# B&R Automation Studio project VisionSample (part 3)

#### brdkFile_func.h - Header for internal functions for library.
```c
#ifndef BRDK_FILE_FUNCS
#define BRDK_FILE_FUNCS 1

#include <brdkFile.h>
#include <bur/plctypes.h>

#ifdef __cplusplus
	extern "C"
	{
#endif

#ifdef __cplusplus
	};
#endif

#define false 0
#define true 1
#define NULL 0

unsigned long buildParameterString(char* pDrive,char* pPath, char* pDeviceParam);
char* getDrive(brdk_file_drive_typ drive, char* pDrive);
signed long splitFolderPath(char* pDestination, char* pSource);

#endif /* !BRDK_FILE_FUNCS */
```

#### brdkFile_func.c - Internal functions for library.
```c
#include <brdkFile_func.h>

unsigned long buildParameterString(char* pDrive,char* pPath, char* pDeviceParam) {
	brdkStrCpy((unsigned long)pDeviceParam,(unsigned long)"/DEVICE=\"");
	brdkStrCat((unsigned long)pDeviceParam,(unsigned long)pDrive);
	brdkStrCat((unsigned long)pDeviceParam,(unsigned long)"\\");
	if(pPath[0] != 0) {
		brdkStrReplace((unsigned long)pPath,(unsigned long)"/",(unsigned long)"\\");	/* replace any front slah with backslash */
		brdkStrCat((unsigned long)pDeviceParam,(unsigned long)pPath);
	}
	brdkStrCat((unsigned long)pDeviceParam,(unsigned long)"\"");
	return (unsigned long)pDeviceParam;
}

char* getDrive(brdk_file_drive_typ drive, char* pDrive) {
	switch(drive) {
		case C_DRIVE: brdkStrCpy((unsigned long)pDrive,(unsigned long)"C:\\"); break;
		case D_DRIVE: brdkStrCpy((unsigned long)pDrive,(unsigned long)"D:\\"); break;
		case E_DRIVE: brdkStrCpy((unsigned long)pDrive,(unsigned long)"E:\\"); break;
		case F_DRIVE: brdkStrCpy((unsigned long)pDrive,(unsigned long)"F:\\"); break;
		case G_DRIVE: brdkStrCpy((unsigned long)pDrive,(unsigned long)"G:\\"); break;
	}
	return pDrive;
}

signed long splitFolderPath(char* pDestination, char* pSource) {
	int idx = 0;
	signed long pos = -1;
	if(pSource[idx] != 0) {
		pos = brdkStrIndexOf((unsigned long)&pSource[idx],(unsigned long)"\\",BRDK_STR_LEFT_SEARCH);
		if(pos > -1) {
			brdkStrMemCpy((unsigned long)pDestination,(unsigned long)&pSource[idx],(unsigned long)++pos);
			pDestination[pos] = 0;
		}
	}
	return pos;
}
```

- CHANGELOG - brdkFile change log file (not shown)

### revision.txt
```
Version 5.26
- Update to mappVision 4.26
- Changed image request to official function block
- Removed recipe management
- Removed color detection
- Removed optic details
- Removed VC4 support
- Removed TCP proxy task
- Removed function to load VA applications
- Removed function to download images

Version 5.24
- Update to AS 4.12
- Update to mapp 4.24
- Fixed image download node number is not correct
- Removed old routing files
- Changed image update interval to 500ms

Version 5.15
- Update recipe managment to V1.0
- Updated constant for code reader parameter "ParameterMode"
- Fix ViColor
- Make it possible to change connections
- Updated to official 5.15 versions and official lightbar upgrade
- Vi_Optics added

Version 2.3
 - Added RouteInfo_Tool.ps1
 - Added color detection first version
 - Split up main task into main and visu, integrated light task into main and visu
 - Added funkctionality to rotate the image on the main page
 - Click on the image on the main page toggles now the textposition (crosshair-details) from left to right
 - CodeReader and OCR Text will be shown on the main page and saved in SVG file
 - Added proxy task to eliminate routing batch file
 - Added Pixel Counter hardware and code

Version 2.2
- Added new functionality to show images in every size on the webviewer widget on the mainpage
- Improved repetitive mode
- SVG files save now all information. It is possible to click on the crosshairs to show the details
- Added diagnostic data creation
- Updated recipe management
- Changed public arrays start index to 0 to avoid issues with C task
- Added a VC4 visualization
- Added functionality to show the image on the VC4 visualization (documentation still missing)
- After boot the first found light will be selected
- Some additional improvements, code optimizations & bug fixes

Version 2.1
- Simplified and reduced data structures
- Added function to switch vision applications
- Reduced result content to one page
- Simplified and sorted the task Vi_image
- Moved crosshair handling to task Vi_image
- Some bugfixes in task Vi_image
- Updated to official versions

Version 2.0
- Convert data structure to new camera firmware
- Support for multiple camera's
- Recipe managment for loading and saving parameters
- Download camera images directly through web browser
- Cleaned up UI
- Support for external lights
- Sample task for nettime with motion
```

### VisionVariables.var
```iecst
(*-----------------------------------------------------------------------------------------------------------------------------------------*)
(*Global variables for sensor hardware and vision functions*)
VAR
	gBlob : typBlobMain; (*Data that is specific for the blob function*)
	gCodeReader : typCodeReaderMain; (*Data that is specific for the code reader*)
	gMatch : typMatchMain; (*Data that is specific for the match function*)
	gMT : typMTMain; (*Data that is specific for the measurement function*)
	gOCR : typOCRMain; (*Data that is specific for the OCR function*)
	gPixel : typPixelMain; (*Data that is specific for the Pixel Counter function*)
	gVisionImage : typVisionImage; (*Data for image handling*)
	gVisionLight : ARRAY[0..MAX_NUM_LIGHTS] OF typLightMain; (*General Light  functions that are independent from the inspection function*)
	gVisionNettime : typVisionNettime; (*Data for nettime calculation*)
	gVisionSensor : ARRAY[0..MAX_NUM_CAMS] OF typVisionMain; (*General vision functions that are independent from the inspection function*)
	gSelectedSensor : UINT := 1; (*Selected camera node number*)
	gSelectedLight : UINT := 1; (*Selected Light node number*)
	NettimeCurrent_us : DINT; (*Current Powerlink nettime*)
END_VAR
(*-----------------------------------------------------------------------------------------------------------------------------------------*)
(*Global constants*)
VAR CONSTANT
	MAX_NUM_CAMS : UINT := 6; (*Maximum number of camera's*)
	MAX_NUM_LIGHTS : UINT := 5; (*Maximum number of light's*)
	MAX_NUM_RESULTS : UINT := 10; (*Maximum number of results*)
	MAX_NUM_PRODUCTS : UINT := 8; (*Maximum number of products for color detection*)
	MAX_IDX_VA_LIST : UINT := 19; (*Maximum number of entrys in the Vision Application list*)
	CONVERT_CYCLES : UINT := 2000;
	DEVICE_NAME : STRING[40] := 'VisionFileDevice'; (*File device where the images and recipes are stored*)
	NETTIME_DEFAULT_DELAY : UDINT := 30000; (*This delay is used when software trigger is used and nettime is enabled*)
	NETTIME_ENABLE : BOOL := FALSE; (*Enable nettime code, this generates the nettime when using manual triggers*)
	MAX_NUM_CODETYPES : USINT := 69; (*Maximum number of code types*)
END_VAR
VAR
	CodeTypes : {REDUND_UNREPLICABLE} ARRAY[0..MAX_NUM_CODETYPES] OF STRING[80] := ['Auto Identify (0)','2/5 Industrial (1)','2/5 Interleaved (2)','Codebar (3)','Code 32 (4)','Code 39 (5)','Code 93 (6)','Code 128 (7)','MSI (8)','PharmaCode (9)','EAN-8 (10)','EAN-8 Add-On 2 (11)','EAN-8 Add-On 5 (12)','EAN-13 (13)','EAN-13 Add-On 2 (14)','EAN-13 Add-On 5 (15)',4(''),'UPC-A (20)','UPC-A Add-On 2 (21)','UPC-A Add-On 5 (22)','UPC-E (23)','UPC-E Add-On 2 (24)','UPC-E Add-On 5 (25)',4(''),'GS1-128 (30)','GS1 DataBar Omnidirectional (31)','GS1 DataBar Truncated (32)','GS1 DataBar Stacked (33)','GS1 DataBar Stacked Omnidirectional (34)','GS1 DataBar Limited (35)','GS1 DataBar Expanded (36)','GS1 DataBar ExpandedStacked (37)',12(''),'Data Matrix ECC200 (50)','QR Code Model 1 (51)','QR Code Model 2 (52)','Micro QRCode (53)','PDF417 (54)','Aztec Code (55)',4(''),'GS1 Data Matrix (60)','GS1 QR Code Model 1 (61)','GS1 QR Code Model 2 (62)','GS1 Aztec Code (63)',6('')]; (*Codes types for code reading*)
END_VAR
```

### VisionTypes.typ
```iecst
(*-----------------------------------------------------------------------------------------------------------------------------------------*)
(*General vision structures*)

TYPE
	typVisionMain : 	STRUCT
		CMD : typVisionCommand;
		CFG : typVisionConfig;
		DAT : typVisionData;
		HW : typVisionHW;
	END_STRUCT;
	typVisionCommand : 	STRUCT
		ImageTrigger : BOOL;
		ImageTriggerReset : BOOL;
		AutoSetupStartStop : BOOL;
	END_STRUCT;
	typVisionConfig : 	STRUCT
		VisionFunction : enumVisionFunction;
		PowerlinkNode : USINT;
		DataStructure : UDINT;
		ComponentLink : ViComponentType;
		ResolutionWidth_X : UINT; (*Nr of sensor pixels in x direction (width). Is always bigger than height*)
		ResolutionHeight_Y : UINT; (*Nr of sensor pixels in y direction (height). Is always smaller than width*)
	END_STRUCT;
	typVisionData : 	STRUCT
		Enable : BOOL := FALSE;
		MaxItemCnt : USINT := 10;
		NettimeDelay : DINT;
		Timeout : UINT := 5000;
		Gain : USINT;
		Focus : UINT;
		Exposure : UDINT;
		FlashColor : USINT := 1;
		FlashSegment : USINT := 15;
		LedColor : USINT;
		IRFilter : BOOL;
		OffsetROIX : DINT;
		OffsetROIY : DINT;
		OffsetROIRotationCenterX : DINT;
		OffsetROIRotationCenterY : DINT;
		OffsetROIOrientation : INT;
		ChromaticLock : BOOL;
		Alignment : USINT;
		AutoSetupGain : USINT;
		AutoSetupFocus : UINT;
		AutoSetupExposure : UDINT;
		AcquisitionAcceptedCnt : USINT;
		AcquisitionCompletedCnt : USINT;
		AcquisitionFailedCnt : USINT;
		LightWarningCnt : USINT;
		ImageProcessingError : UINT;
		ImageProcessingActive : BOOL;
		ImageNettime : DINT;
		ProcessingTimeCamera : UINT;
		ProcessingTimeFunction : UINT;
		ResultCnt : USINT;
		CockpitIsActive : BOOL;
		Status : UDINT;
		StatusText : STRING[30];
		Active : BOOL;
	END_STRUCT;
	typVisionHW : 	STRUCT
		Connected : BOOL;
		Ready : BOOL;
		DigitalInput01 : BOOL;
		DigitalOutput01 : BOOL;
		DigitalOutputStatus01 : BOOL;
		DigitalOutput02 : BOOL;
		DigitalOutputStatus02 : BOOL;
		SerialNumber : UDINT;
		ID : UDINT;
		Variant : UDINT;
		Firmware : UDINT;
		Undervoltage : BOOL;
		Temperature : SINT;
	END_STRUCT;
	enumVisionFunction :
		(
		enumFunctionNone,
		enumBlob,
		enumCoderReader,
		enumMatch,
		enumMeasurement,
		enumOCR,
		enumPixelCounter
		);
END_TYPE

(*-----------------------------------------------------------------------------------------------------------------------------------------*)
(*General Light structures*)

TYPE
	typLightMain : 	STRUCT
		CMD : typLightCommand;
		CFG : typLightConfig;
		DAT : typLightData;
		HW : typLightHW;
	END_STRUCT;
	typLightCommand : 	STRUCT
		FlashTrigger : BOOL;
		FlashTriggerReset : BOOL;
	END_STRUCT;
	typLightConfig : 	STRUCT
		LightType : enumLightType;
		PowerlinkNode : USINT;
	END_STRUCT;
	typLightData : 	STRUCT
		Enable : USINT := 1;
		FlashColor : USINT := 1;
		FlashSegment : UINT := 15;
		Exposure : UDINT := 200;
		SetAngle : UINT;
		Timeout : UINT := 5000;
		NettimeDelay : DINT;
		FlashAcceptedCnt : USINT;
		FlashCompletedCnt : USINT;
		FlashFailedCnt : USINT;
		Status : UDINT;
	END_STRUCT;
	typLightHW : 	STRUCT
		Connected : BOOL;
		Ready : BOOL;
		SerialNumber : UDINT;
		ID : UDINT;
		Variant : UDINT;
		Firmware : UDINT;
		TemperatureLED : SINT;
		TemperatureControllerBoard : SINT;
		WarningCnt : USINT;
	END_STRUCT;
	enumLightType :
		(
		enumLightNone,
		enumBacklight,
		enumLightbar
		);
END_TYPE

(*-----------------------------------------------------------------------------------------------------------------------------------------*)
(*General nettime structures*)

TYPE
	typVisionNettime : 	STRUCT
		CMD : typNettimeCommand;
		CFG : typNettimeConfig;
		DAT : typNettimeData;
	END_STRUCT;
	typNettimeCommand : 	STRUCT
		Activate : BOOL;
	END_STRUCT;
	typNettimeConfig : 	STRUCT
		AxisPeriod : LREAL; (*Units when period repeats*)
		AxisPositionTrigger : LREAL; (*Position in the period where trigger is fired*)
		AxisPositionDelay_Cycles : LREAL; (*Delay in PLK cycles for the read position from drive*)
		VisionPreTrigger_Cycles : DINT; (*Number of powerlink cycles the trigger has to be send ahead*)
	END_STRUCT;
	typNettimeData : 	STRUCT
		NettimeNext_us : DINT; (*Calculated nettime for next trigger*)
		NettimeDelta_us : DINT; (*Difference between current nettime and calculated nettime for the camera trigger*)
		AxisPosition : LREAL; (*Current axis position*)
		AxisVelocity : LREAL; (*Current axis position*)
		AxisInVelocity : BOOL; (*Indicates that the axis is moving at speed*)
		Overflow : DINT; (*Counts up when a trigger could not be set on time*)
	END_STRUCT;
END_TYPE

(*-----------------------------------------------------------------------------------------------------------------------------------------*)
(*Image upload structures*)

TYPE
	typVisionImage : 	STRUCT
		CMD : typVisionImageCommand;
		CFG : typVisionImageConfig;
		DAT : typVisionImageData;
	END_STRUCT;
	typVisionImageCommand : 	STRUCT
		CreateDir : BOOL;
		DeleteDir : BOOL;
		DeleteImage : BOOL;
		GetImage : BOOL;
		SaveImage : BOOL;
		Refresh : BOOL;
		ResetError : BOOL;
	END_STRUCT;
	typVisionImageConfig : 	STRUCT
		FileDevice : STRING[80];
		FileName : STRING[80];
		DirName : STRING[80];
		ComponentLink : ViComponentType;
	END_STRUCT;
	typVisionImageData : 	STRUCT
		ImagesList : ARRAY[0..19]OF STRING[80];
		ImageSelected : STRING[80];
		ImagePath : STRING[80];
		ImageLast : STRING[80];
		Crosshair : ARRAY[1..MAX_NUM_RESULTS]OF typVisionImageDataCrosshair;
		Status : DINT;
	END_STRUCT;
	typVisionImageDataCrosshair : 	STRUCT
		CrosshairX : REAL;
		CrosshairY : REAL;
		CrosshairRotate : REAL;
		Text : STRING[1000];
	END_STRUCT;
END_TYPE

(*-----------------------------------------------------------------------------------------------------------------------------------------*)
(*Vision specific structures*)

TYPE
	typCodeReaderMain : 	STRUCT  (*Code reader structures*)
		CodeType : USINT;
		GradingEnable : BOOL;
		RobustnessEnable : BOOL;
		ParameterMode : USINT;
		ParameterOptimization : USINT;
		BarcodeText : ARRAY[1..MAX_NUM_RESULTS]OF STRING[100];
		BarcodeType : ARRAY[1..MAX_NUM_RESULTS]OF USINT;
		PositionX : ARRAY[1..MAX_NUM_RESULTS]OF DINT;
		PositionY : ARRAY[1..MAX_NUM_RESULTS]OF DINT;
		Orientation : ARRAY[1..MAX_NUM_RESULTS]OF INT;
		Grading : ARRAY[1..MAX_NUM_RESULTS]OF SINT;
		EnhancedGrading : ARRAY[1..23]OF USINT;
	END_STRUCT;
	typBlobMain : 	STRUCT  (*Blob function structures*)
		RegionalFeature : BOOL;
		EnhancedBlobInformation : BOOL := FALSE;
		ModelNumber : ARRAY[1..MAX_NUM_RESULTS]OF USINT;
		Clipped : ARRAY[1..MAX_NUM_RESULTS]OF BOOL;
		Area : ARRAY[1..MAX_NUM_RESULTS]OF UDINT;
		PositionX : ARRAY[1..MAX_NUM_RESULTS]OF DINT;
		PositionY : ARRAY[1..MAX_NUM_RESULTS]OF DINT;
		Orientation : ARRAY[1..MAX_NUM_RESULTS]OF INT;
		MeanGrayValue : ARRAY[1..MAX_NUM_RESULTS]OF USINT;
		Length : ARRAY[1..MAX_NUM_RESULTS]OF UDINT;
		Width : ARRAY[1..MAX_NUM_RESULTS]OF UDINT;
	END_STRUCT;
	typMatchMain : 	STRUCT  (*Match function structures*)
		MinScore : USINT := 70;
		MaxOverlap : USINT;
		ModelNumber : ARRAY[1..MAX_NUM_RESULTS]OF USINT;
		Score : ARRAY[1..MAX_NUM_RESULTS]OF USINT;
		PositionX : ARRAY[1..MAX_NUM_RESULTS]OF DINT;
		PositionY : ARRAY[1..MAX_NUM_RESULTS]OF DINT;
		Orientation : ARRAY[1..MAX_NUM_RESULTS]OF INT;
		Scale : ARRAY[1..MAX_NUM_RESULTS]OF USINT;
		RotCenterX : ARRAY[1..MAX_NUM_RESULTS]OF DINT;
		RotCenterY : ARRAY[1..MAX_NUM_RESULTS]OF DINT;
	END_STRUCT;
	typOCRMain : 	STRUCT  (*OCR function structures*)
		ParameterMode : USINT;
		GradingEnable : BOOL;
		Text : ARRAY[1..MAX_NUM_RESULTS]OF STRING[50];
		Grading : ARRAY[1..MAX_NUM_RESULTS]OF USINT;
		PositionX : ARRAY[1..MAX_NUM_RESULTS]OF DINT;
		PositionY : ARRAY[1..MAX_NUM_RESULTS]OF DINT;
		Orientation : ARRAY[1..MAX_NUM_RESULTS]OF INT;
	END_STRUCT;
	typPixelMain : 	STRUCT  (*OCR function structures*)
		EnhancedPixelCounterInformation : BOOL := FALSE;
		ModelNumber : ARRAY[1..MAX_NUM_RESULTS]OF USINT;
		NumPixels : ARRAY[1..MAX_NUM_RESULTS]OF UDINT;
		MinGray : ARRAY[1..MAX_NUM_RESULTS]OF USINT;
		MaxGray : ARRAY[1..MAX_NUM_RESULTS]OF USINT;
		MeanGray : ARRAY[1..MAX_NUM_RESULTS]OF UINT;
		DeviationGray : ARRAY[1..MAX_NUM_RESULTS]OF UINT;
		MedianGray : ARRAY[1..MAX_NUM_RESULTS]OF USINT;
		ModelArea : ARRAY[1..MAX_NUM_RESULTS]OF UDINT;
		NumConnectedComponents : ARRAY[1..MAX_NUM_RESULTS]OF UINT;
		PositionX : ARRAY[1..MAX_NUM_RESULTS]OF DINT;
		PositionY : ARRAY[1..MAX_NUM_RESULTS]OF DINT;
	END_STRUCT;
	typMTMain : 	STRUCT  (*MT function structures*)
		UseResultAsXY : BOOL;
		ParameterMode : USINT;
		Result : ARRAY[1..MAX_NUM_RESULTS]OF DINT;
	END_STRUCT;
END_TYPE
```

### Program Logical/Vision/Vi_main (IEC)

#### Main.st - Init, cyclic, exit code
```iecst
// --------------------------------------------------------------------------------------------------------------------
// General vision task. This is a support task for the mappVision. The following functions are implemneted
// - Translate some values in text messages
// - Reset camera trigger when inspection is finsihed
// - Load vision application
// - Save diagnostic data
// Version 2.x (Check revision history for details)
// --------------------------------------------------------------------------------------------------------------------
PROGRAM _INIT

END_PROGRAM

// -----------------------------------------------------------------------------------------------------------
// Cyclic part
// -----------------------------------------------------------------------------------------------------------
PROGRAM _CYCLIC
	// -----------------------------------------------------------------------------------------------------------
	// Translate camera status in readable text
	// -----------------------------------------------------------------------------------------------------------
	IF gVisionSensor[idSensor].DAT.Status = 0 THEN
		gVisionSensor[idSensor].DAT.StatusText := 'Ready';
	ELSIF gVisionSensor[idSensor].DAT.Status = 16#00000001 THEN
		gVisionSensor[idSensor].DAT.StatusText := 'Image acquisition';
	ELSIF gVisionSensor[idSensor].DAT.Status = 16#00000002 THEN
		gVisionSensor[idSensor].DAT.StatusText := 'Waiting trigger';
	ELSIF gVisionSensor[idSensor].DAT.Status = 16#00000010 THEN
		gVisionSensor[idSensor].DAT.StatusText := 'Searching settings';
	ELSIF gVisionSensor[idSensor].DAT.Status = 16#00000080 THEN
		gVisionSensor[idSensor].DAT.StatusText := 'Setting focus';
	ELSIF gVisionSensor[idSensor].DAT.Status = 16#00000090 THEN
		gVisionSensor[idSensor].DAT.StatusText := 'Searching settings';
	ELSIF gVisionSensor[idSensor].DAT.Status = 16#00000800 THEN
		gVisionSensor[idSensor].DAT.StatusText := 'Cam CPU not ready';
	ELSIF gVisionSensor[idSensor].DAT.Status = 16#00001000 THEN
		gVisionSensor[idSensor].DAT.StatusText := 'Cam sensor not ready';
	ELSIF gVisionSensor[idSensor].DAT.Status = 16#01000000 OR gVisionSensor[idSensor].DAT.Status = 16#02000000 OR gVisionSensor[idSensor].DAT.Status = 16#03000000 THEN
		gVisionSensor[idSensor].DAT.StatusText := 'OS check/update';
	ELSIF gVisionSensor[idSensor].DAT.Status = 16#80000000 THEN
		gVisionSensor[idSensor].DAT.StatusText := 'Vision cockpit active';
	ELSE
		// Display the status in hex format 0x02000800
		gVisionSensor[idSensor].DAT.StatusText := '';
		FOR i := 0 TO 28 BY 4 DO
			gVisionSensor[idSensor].DAT.StatusText := CONCAT(MID(HexTab, 1, LIMIT(1, UDINT_TO_INT((SHR(gVisionSensor[idSensor].DAT.Status, i) AND 16#0000000F) + 1), 16)), gVisionSensor[idSensor].DAT.StatusText);
		END_FOR
		gVisionSensor[idSensor].DAT.StatusText := CONCAT('0x', gVisionSensor[idSensor].DAT.StatusText);
	END_IF

	// -----------------------------------------------------------------------------------------------------------
	// Check if vision cockpit is open
	// -----------------------------------------------------------------------------------------------------------
	gVisionSensor[idSensor].DAT.CockpitIsActive := (gVisionSensor[idSensor].DAT.Status AND 16#8000_0000) > 0;

	// -----------------------------------------------------------------------------------------------------------
	// Auto setup handling
	// -----------------------------------------------------------------------------------------------------------
	IF(gVisionSensor[idSensor].CMD.AutoSetupStartStop AND gVisionSensor[idSensor].DAT.Status <> 0) THEN
		AutoSetupRunning[idSensor] := TRUE;
	ELSIF NOT gVisionSensor[idSensor].CMD.AutoSetupStartStop THEN
		AutoSetupRunning[idSensor] := FALSE;
	END_IF
	IF(gVisionSensor[idSensor].CMD.AutoSetupStartStop AND gVisionSensor[idSensor].DAT.Status = 0 AND AutoSetupRunning[idSensor]) THEN // Setup successfully finished
		gVisionSensor[idSensor].DAT.Gain					:= gVisionSensor[idSensor].DAT.AutoSetupGain;
		gVisionSensor[idSensor].DAT.Focus				:= gVisionSensor[idSensor].DAT.AutoSetupFocus;
		gVisionSensor[idSensor].DAT.Exposure				:= gVisionSensor[idSensor].DAT.AutoSetupExposure;
		gVisionSensor[idSensor].CMD.AutoSetupStartStop	:= FALSE;
		AutoSetupRunning[idSensor]						:= FALSE;
		TON_DelayAfterAutoSetup[idSensor].IN					:= TRUE;
	END_IF
	TON_DelayAfterAutoSetup[idSensor](PT := T#50ms);
	IF TON_DelayAfterAutoSetup[idSensor].Q THEN // After the camera tells it is ready, we need to wait still at least ca 20ms, otherwise it does not accept the trigger
		TON_DelayAfterAutoSetup[idSensor].IN := FALSE;
		IF gVisionSensor[idSensor].HW.Ready AND NOT gVisionSensor[idSensor].DAT.ImageProcessingActive THEN
			IF NETTIME_ENABLE THEN
				gVisionSensor[idSensor].DAT.NettimeDelay := NettimeCurrent_us + NETTIME_DEFAULT_DELAY;
			END_IF
			gVisionSensor[idSensor].CMD.ImageTrigger	:= TRUE;
			gVisionSensor[idSensor].DAT.Active			:= TRUE;
		END_IF
	END_IF

	// -----------------------------------------------------------------------------------------------------------
	// Reset image trigger, reload web page and store image when process is finished
	// -----------------------------------------------------------------------------------------------------------
	IF ((gVisionSensor[idSensor].DAT.AcquisitionCompletedCnt <> AcquisitionCompletedCntOld[idSensor] OR gVisionSensor[idSensor].DAT.AcquisitionFailedCnt <> AcquisitionFailedCntOld[idSensor]) AND NOT gVisionSensor[idSensor].DAT.ImageProcessingActive AND gVisionSensor[idSensor].HW.Ready) THEN
		AcquisitionCompletedCntOld[idSensor]		:= gVisionSensor[idSensor].DAT.AcquisitionCompletedCnt;
		AcquisitionFailedCntOld[idSensor]			:= gVisionSensor[idSensor].DAT.AcquisitionFailedCnt;
		gVisionSensor[idSensor].CMD.ImageTrigger	:= FALSE;
		gVisionSensor[idSensor].DAT.Active			:= FALSE;
	END_IF

	// -----------------------------------------------------------------------------------------------------------
	// Reset trigger when timed out
	// -----------------------------------------------------------------------------------------------------------
	IF gVisionSensor[idSensor].CMD.ImageTrigger THEN
		TriggerTimeoutSensor[idSensor].IN := TRUE;
		TriggerTimeoutSensor[idSensor].PT := REAL_TO_TIME(gVisionSensor[idSensor].DAT.Timeout * 1.25);
		IF TriggerTimeoutSensor[idSensor].Q THEN
			gVisionSensor[idSensor].CMD.ImageTrigger		:= FALSE;
			gVisionSensor[idSensor].CMD.ImageTriggerReset	:= TRUE;
			gVisionSensor[idSensor].DAT.Active				:= FALSE;
		END_IF
	ELSE
		TriggerTimeoutSensor[idSensor].IN := FALSE;
		gVisionSensor[idSensor].CMD.ImageTriggerReset := FALSE;
	END_IF
	TriggerTimeoutSensor[idSensor]();

	// Proceed with next sensor
	idSensor := idSensor + 1;
	IF (idSensor > MAX_NUM_CAMS) THEN
		idSensor := 1;
	END_IF

	// -----------------------------------------------------------------------------------------------------------
	// Reset Light trigger
	// -----------------------------------------------------------------------------------------------------------
	IF (gVisionLight[idLight].DAT.FlashCompletedCnt <> FlashCompletedCntOld[idLight] OR gVisionLight[idLight].DAT.FlashFailedCnt <> FlashFailedCntOld[idLight]) THEN
		FlashCompletedCntOld[idLight]			:= gVisionLight[idLight].DAT.FlashCompletedCnt;
		FlashFailedCntOld[idLight]				:= gVisionLight[idLight].DAT.FlashFailedCnt;
		gVisionLight[idLight].CMD.FlashTrigger	:= FALSE;
	END_IF

	// -----------------------------------------------------------------------------------------------------------
	// Reset trigger when timed out
	// -----------------------------------------------------------------------------------------------------------
	IF gVisionLight[idLight].CMD.FlashTrigger THEN
		TriggerTimeoutLight[idLight].IN := TRUE;
		TriggerTimeoutLight[idLight].PT := REAL_TO_TIME(gVisionLight[idLight].DAT.Timeout * 1.25);
		IF TriggerTimeoutLight[idLight].Q THEN
			gVisionLight[idLight].CMD.FlashTrigger		:= FALSE;
			gVisionLight[idLight].CMD.FlashTriggerReset	:= TRUE;
		END_IF
	ELSE
		TriggerTimeoutLight[idLight].IN := FALSE;
		gVisionLight[idLight].CMD.FlashTriggerReset := FALSE;
	END_IF
	TriggerTimeoutLight[idLight]();

	// Proceed with next light
	idLight := idLight + 1;
	IF (idLight > MAX_NUM_LIGHTS) THEN
		idLight := 1;
	END_IF

END_PROGRAM
```

#### Variables.var - Local variables
```iecst
VAR
	i : UINT;
END_VAR
(*-----------------------------------------------------------------------------------------------------------------------------------------*)
(*Local variables*)
VAR
	idSensor : UINT := 1;
	idLight : UINT := 1;
	TriggerTimeoutSensor : ARRAY[1..MAX_NUM_CAMS] OF TON; (*Disable web reload when timed out*)
	TriggerTimeoutLight : ARRAY[1..MAX_NUM_LIGHTS] OF TON; (*Disable web reload when timed out*)
	AcquisitionFailedCntOld : ARRAY[1..MAX_NUM_CAMS] OF UDINT; (*Old aquisition failed counter*)
	AcquisitionCompletedCntOld : ARRAY[1..MAX_NUM_CAMS] OF UDINT; (*Old aquisition completed counter*)
	AutoSetupRunning : ARRAY[1..MAX_NUM_CAMS] OF BOOL; (*Flag for auto setup running*)
	FlashFailedCntOld : ARRAY[1..MAX_NUM_LIGHTS] OF USINT;
	FlashCompletedCntOld : ARRAY[1..MAX_NUM_LIGHTS] OF USINT;
END_VAR
VAR CONSTANT
	HexTab : STRING[16] := '0123456789ABCDEF';
END_VAR
VAR
	TON_DelayAfterAutoSetup : ARRAY[1..MAX_NUM_CAMS] OF TON;
END_VAR
```

#### Types.typ
```iecst
TYPE
	local_axisTrig_typ : 	STRUCT
		nettimeLastCycle_us : DINT;
		powerlinkCycle_us : DINT;
		axisPositionNow : REAL;
		triggerPosDelta : REAL;
		triggerTimeDelta : DINT; (*In us*)
	END_STRUCT;
	local_typ : 	STRUCT
		path : STRING[100];
		brdkViBase_imgTrigger_0 : brdkViBase_imgTrigger;
		brdkViBase_getCameraInfo_0 : brdkViBase_getCameraInfo;
		mappView : {REDUND_UNREPLICABLE} brdkViImg_mappView;
		viBaseSaveDiagData_0 : ViBaseSaveDiagData;
		fileDelete : FileDelete;
		visionDiagFileDevice : STRING[10];
		viBaseLoadApplication_0 : ViBaseLoadApplication;
		axisTrig : local_axisTrig_typ;
		brdkFileWrite : brdkFileWrite;
		dtNow : DTStructure;
		DTGetTime_0 : DTGetTime;
		tmp2D : brdkViBase_2d_typ;
		strElemId : STRING[80];
		oldIntElemID : USINT;
		elemId : STRING[80];
	END_STRUCT;
	hmi_typ : 	STRUCT
		in : hmi_in_typ;
		out : hmi_out_typ;
	END_STRUCT;
	hmi_out_vf_typ : 	STRUCT
		processingTime : UDINT;
		numResults : USINT;
		crData : ARRAY[0..9]OF STRING[240];
		match : typMatchMain;
		measurement : typMTMain;
		codeReader : typCodeReaderMain;
		ocr : typOCRMain;
		pixelCnt : typPixelMain;
		blob : typBlobMain;
		ocrData : ARRAY[0..9]OF STRING[240];
	END_STRUCT;
	hmi_out_lights_typ : 	STRUCT
		status : brdkViBase_light_hw_status_typ;
		common : brdkViBase_hw_in_common_typ;
		simulated : BOOL;
		connectedText : STRING[20];
		connected : BOOL;
		mappVisionActive : BOOL;
		processing : BOOL;
		ready : BOOL;
		statusText : STRING[50];
		lightType : STRING[20];
		plNodeNr : USINT;
	END_STRUCT;
	hmi_out_camera_typ : 	STRUCT
		simulated : BOOL;
		connectedText : STRING[20];
		connected : BOOL;
		mappVisionActive : BOOL;
		processing : BOOL;
		ready : BOOL;
		statusText : STRING[50];
		plNodeNr : USINT;
		visionFunction : STRING[20];
		processingTime : UDINT;
		opticInfo : brdkViBase_opticInfo_typ;
		common : brdkViBase_hw_in_common_typ;
		hw : brdkViBase_cam_hw_in_status_typ;
	END_STRUCT;
	hmi_out_typ : 	STRUCT
		svgOverlay : STRING[10000];
		wsPort : UINT;
		lights : ARRAY[START_IDX..NUM_LIGHTS]OF hmi_out_lights_typ;
		camera : hmi_out_camera_typ;
		VF : hmi_out_vf_typ;
		status : DINT;
	END_STRUCT;
	hmi_in_cmd_flashSegment_typ : 	STRUCT
		top : BOOL := TRUE;
		bottom : BOOL := TRUE;
		right : BOOL := TRUE;
		left : BOOL := TRUE;
	END_STRUCT;
	hmi_in_cmd_typ : 	STRUCT
		lights : ARRAY[START_IDX..NUM_LIGHTS]OF brdkViBase_light_hw_out_cmd_typ;
		flashSegment : hmi_in_cmd_flashSegment_typ;
		repetitiveTrigger : BOOL; (*Enable Repetitive trigger*)
		trigger : BOOL; (*Trigger a image*)
		autoSearch : BOOL; (*Start auto Search of exposure and focus for camra*)
		resetInfo : BOOL; (*Reset optic info to the current camera*)
		saveDiagnositc : BOOL; (*Save vision diagnostic *)
		loadVA : BOOL; (*Load Vision application*)
		saveImage : BOOL;
		intElemId : USINT := 1;
		elemId : STRING[80];
		click : BOOL;
		y : REAL;
		x : REAL;
		shapeSelector : ARRAY[0..2]OF STRING[100] := ['{"value":"1", "text":"Rectangle"}','{"value":"2", "text":"Circle"}','{"value":"3", "text":"Triangle"}'];
		strokeColorSelector : ARRAY[0..5]OF STRING[100] := ['{"value":";stroke:black", "text":"Black"}','{"value":";stroke:white", "text":"White"}','{"value":";stroke:red", "text":"Red"}','{"value":";stroke:green", "text":"Green"}','{"value":";stroke:blue", "text":"Blue"}','{"value":";stroke:yellow", "text":"Yellow"}'];
		fillColorSelector : ARRAY[0..5]OF STRING[100] := ['{"value":"fill:black", "text":"Black"}','{"value":"fill:white", "text":"White"}','{"value":"fill:red", "text":"Red"}','{"value":"fill:green", "text":"Green"}','{"value":"fill:blue", "text":"Blue"}','{"value":"fill:yellow", "text":"Yellow"}'];
		draw : hmi_in_cmd_draw_typ;
	END_STRUCT;
	hmi_in_cmd_draw_typ : 	STRUCT
		intShape : INT; (*0 = rectangle, 1 = circle, 2 = triangle*)
		radius : REAL := 60;
		width : REAL := 80;
		length : REAL := 80;
		invRotation : REAL;
		rotation : REAL;
		strFillColor : STRING[80];
		strStrokeColor : STRING[80];
		strStrokeWidth : STRING[80];
		strFillOpac : STRING[80];
		strStrokeOpac : STRING[80];
		intStrokeWidth : INT := 6;
		realFillOpac : REAL := 0;
		realStrokeOpac : REAL := 1;
		strStyleHighlight : STRING[240];
		strStyle : STRING[240];
	END_STRUCT;
	hmi_in_typ : 	STRUCT
		cmd : hmi_in_cmd_typ;
		recipe : recipe_typ;
		cameraInfo : brdkViBase_camInfo_typ;
		diagnosticFilename : STRING[50];
		vaName : STRING[50];
		lightNum : USINT := 1;
	END_STRUCT;
	hw_io_in_typ : 	STRUCT
		nettime : DINT;
	END_STRUCT;
	hw_io_typ : 	STRUCT
		in : hw_io_in_typ;
	END_STRUCT;
	hw_typ : 	STRUCT
		camera : brdkViBase_cam_hw_typ;
		VF : hw_VF_typ;
		lights : ARRAY[START_IDX..NUM_LIGHTS]OF brdkViBase_light_hw_typ;
		io : hw_io_typ;
	END_STRUCT;
	hw_VF_typ : 	STRUCT
		codeReader : brdkViBase_hw_cr_10_typ;
		pixelCnt : brdkViBase_hw_pxCnt_10_typ;
		measurement : brdkViBase_hw_mes_10_typ;
		matching : brdkViBase_hw_match_10_typ;
		ocr : brdkViBase_hw_OCR_10_typ;
		blob : brdkViBase_hw_blob_10_typ;
	END_STRUCT;
	recipe_typ : 	STRUCT
		lights : ARRAY[START_IDX..NUM_LIGHTS]OF brdkViBase_light_hw_out_par_typ;
		cam : brdkViBase_cam_recipe_typ;
		BLOB : brdkViBase_hw_blob_out_typ;
		CR : brdkViBase_hw_cr_out_typ;
		match : brdkViBase_hw_match_out_typ;
		meassurement : brdkViBase_hw_mes_out_typ;
		OCR : brdkViBase_hw_OCR_out_typ;
		pxCnt : brdkViBase_hw_pxCnt_out_typ;
	END_STRUCT;
	common_recipe_typ : 	STRUCT
		jpegQuality : USINT;
		imageFormat : BRDKVIIMG_IMG_TYPE;
		visionPreTriggerCycles : DINT := 0;
		enableAxisTrigger : BOOL;
	END_STRUCT;
END_TYPE
```

#### Variables1.var
```iecst
VAR
	tmpID : STRING[80];
	tmpVF : STRING[80];
	tmpStr : STRING[100];
	commonRecipe : common_recipe_typ;
END_VAR
VAR CONSTANT
	START_IDX : USINT := 1;
END_VAR
VAR
	p : USINT;
	tableNo : ARRAY[1..10] OF BYTE;
	MAX_NUM_RESULTS : USINT;
END_VAR
VAR CONSTANT
	NUM_LIGHTS : USINT := 9;
END_VAR
VAR
	debug : BOOL;
END_VAR
VAR CONSTANT
	NUM_CAMS : USINT := 6;
END_VAR
VAR
	this : REFERENCE TO local_typ;
	hmi : REFERENCE TO hmi_typ;
	hw : REFERENCE TO hw_typ;
	hmiInstance : ARRAY[START_IDX..NUM_CAMS] OF hmi_typ;
	hwInstance : ARRAY[START_IDX..NUM_CAMS] OF hw_typ;
	localInstance : ARRAY[START_IDX..NUM_CAMS] OF local_typ;
	watchIdx : USINT;
	k : USINT;
	j : USINT;
	u : USINT;
	idx : USINT;
END_VAR
```

#### hmiAction.st
```iecst
ACTION hmiAction:

	IF DiagCpuIsSimulated() OR (NOT hw.camera.in.common.moduleOk AND this.brdkViBase_imgTrigger_0.simulate.alwaysSimulateNonePresentCamera) THEN
		hmi.out.camera.connected :=  TRUE;
		hmi.out.camera.simulated := TRUE;
	ELSE

		hmi.out.camera.simulated := FALSE;
		IF hw.camera.in.common.moduleOk THEN
			hmi.out.camera.connected :=  TRUE;
		ELSE
			hmi.out.camera.connected :=  FALSE;
		END_IF
	END_IF
	hmi.out.camera.processing := hw.camera.in.status.imageProcessingActive;
	hmi.out.camera.ready := this.brdkViBase_imgTrigger_0.ready AND NOT hmi.in.cmd.repetitiveTrigger;

	brsmemcpy(ADR(hmi.out.camera.hw),ADR(hw.camera.in.status),SIZEOF(hmi.out.camera.hw));
	brsmemcpy(ADR(hmi.out.camera.common),ADR(hw.camera.in.common),SIZEOF(hmi.out.camera.common));

	hmi.in.recipe.cam.flashSegment.0 := hmi.in.cmd.flashSegment.top;
	hmi.in.recipe.cam.flashSegment.1 := hmi.in.cmd.flashSegment.bottom;
	hmi.in.recipe.cam.flashSegment.2 := hmi.in.cmd.flashSegment.left;
	hmi.in.recipe.cam.flashSegment.3 := hmi.in.cmd.flashSegment.right;

	FOR i:=START_IDX TO NUM_LIGHTS DO
		hmi.out.lights[i].common:=hw.lights[i].in.common;
		hmi.out.lights[i].status:=hw.lights[i].in.status;
	END_FOR;
END_ACTION
```

#### processResultsAction.st
```iecst
ACTION processResultsAction:

	//Conversion of individual USINT values into strings for OCR
	brsmemset(ADR(hmi.out.VF.ocrData),0,SIZEOF(hmi.out.VF.ocrData));
	IF  hw.VF.ocr.in.common.numResults > 0 THEN
		FOR j:=0 TO hw.VF.ocr.in.common.numResults-1 DO
			brsmemcpy(ADR(hmi.out.VF.ocrData[j]),ADR(hw.VF.ocr.in.results[j].data),SIZEOF(hw.VF.ocr.in.results[j].data));
		END_FOR;
	END_IF

	//Conversion of individual USINT values into strings for Code Reader
	brsmemset(ADR(hmi.out.VF.crData),0,SIZEOF(hmi.out.VF.crData));
	IF  hw.VF.codeReader.in.common.numResults > 0 THEN
		FOR j:=0 TO hw.VF.codeReader.in.common.numResults-1 DO
			brsmemcpy(ADR(hmi.out.VF.crData[j]),ADR(hw.VF.codeReader.in.results[j].data),SIZEOF(hw.VF.codeReader.in.results[j].data));
		END_FOR;
	END_IF

	// conversion of variables to suitable data types
	hmi.in.cmd.draw.strStrokeWidth := INT_TO_STRING(hmi.in.cmd.draw.intStrokeWidth);
	hmi.in.cmd.draw.strFillOpac := REAL_TO_STRING(hmi.in.cmd.draw.realFillOpac);
	hmi.in.cmd.draw.strStrokeOpac := REAL_TO_STRING(hmi.in.cmd.draw.realStrokeOpac);

	hmi.in.cmd.draw.invRotation:= -(hmi.in.cmd.draw.rotation);

	// DRAW CIRCLES ON RESULTS
	hmi.out.svgOverlay := '';
	//BLOB
	IF hw.VF.blob.in.common.numResults > 0 THEN

		FOR i:= 1 TO hw.VF.blob.in.common.numResults BY 1 DO
			this.tmp2D.x := DINT_TO_REAL(hw.VF.blob.in.results[i-1].positionX) / 100.0;
			this.tmp2D.y := DINT_TO_REAL(hw.VF.blob.in.results[i-1].positionY) / 100.0;

			// Style string generation
			// e.g.:'id="13" style="fill:blue;stroke:blue;stroke-width:5;fill-opacity:0.3;stroke-opacity:1"'

			this.strElemId := UINT_TO_STRING(i);

			hmi.in.cmd.draw.strStyle := 'id="1';

			styleStringGeneration;

			// Draw selested shape with specified parameters on the overlay
			CASE hmi.in.cmd.draw.intShape OF
				0: // Rectangle
					brdkViGeom_drawSvgRectFromCP(this.tmp2D,hmi.in.cmd.draw.length,hmi.in.cmd.draw.width,hmi.in.cmd.draw.invRotation,ADR(hmi.out.svgOverlay),ADR(hmi.in.cmd.draw.strStyle));
				1: // Circle
					brdkViGeom_drawSvgCircle(this.tmp2D,hmi.in.cmd.draw.radius,ADR(hmi.out.svgOverlay),ADR(hmi.in.cmd.draw.strStyle));
				2: // Triangle
					brdkViGeom_drawSvgTriFromCP(this.tmp2D,hmi.in.cmd.draw.length,hmi.in.cmd.draw.width,hmi.in.cmd.draw.invRotation,ADR(hmi.out.svgOverlay),ADR(hmi.in.cmd.draw.strStyle));
			END_CASE;
		END_FOR;
	END_IF;

	//CODE READER

	IF hw.VF.codeReader.in.common.numResults > 0 THEN

		hmi.out.svgOverlay := '';

		FOR i:= 1 TO hw.VF.codeReader.in.common.numResults BY 1 DO
			this.tmp2D.x := DINT_TO_REAL(hw.VF.codeReader.in.results[i-1].positionX) / 100.0;
			this.tmp2D.y := DINT_TO_REAL(hw.VF.codeReader.in.results[i-1].positionY) / 100.0;

			// Style string generation
			// e.g.:'id="13" style="fill:blue;stroke:blue;stroke-width:5;fill-opacity:0.3;stroke-opacity:1"'

			this.strElemId := UINT_TO_STRING(i);

			hmi.in.cmd.draw.strStyle := 'id="2';

			styleStringGeneration;

			hmi.in.cmd.draw.rotation:= hw.VF.codeReader.in.results[i-1].orientation / 100.0;
			hmi.in.cmd.draw.invRotation:= -(hmi.in.cmd.draw.rotation);

			// DRAW SELECTED SHAPE WITH SPECIFIED PARAMETERS ON THE OVERLAY
			CASE hmi.in.cmd.draw.intShape OF
				0: // Rectangle
					brdkViGeom_drawSvgRectFromCP(this.tmp2D,hmi.in.cmd.draw.length,hmi.in.cmd.draw.width,hmi.in.cmd.draw.invRotation,ADR(hmi.out.svgOverlay),ADR(hmi.in.cmd.draw.strStyle));
				1: // Circle
					brdkViGeom_drawSvgCircle(this.tmp2D,hmi.in.cmd.draw.radius,ADR(hmi.out.svgOverlay),ADR(hmi.in.cmd.draw.strStyle));
				2: // Triangle
					brdkViGeom_drawSvgTriFromCP(this.tmp2D,hmi.in.cmd.draw.length,hmi.in.cmd.draw.width,hmi.in.cmd.draw.invRotation,ADR(hmi.out.svgOverlay),ADR(hmi.in.cmd.draw.strStyle));

			END_CASE;
		END_FOR;
	END_IF;

	//MATCHING

	IF hw.VF.matching.in.common.numResults > 0 THEN

		hmi.out.svgOverlay := '';

		FOR i:= 1 TO hw.VF.matching.in.common.numResults BY 1 DO
			this.tmp2D.x := DINT_TO_REAL(hw.VF.matching.in.results[i-1].positionX) / 100.0;
			this.tmp2D.y := DINT_TO_REAL(hw.VF.matching.in.results[i-1].positionY) / 100.0;

			// Style string generation
			// e.g.:'id="13" style="fill:blue;stroke:blue;stroke-width:5;fill-opacity:0.3;stroke-opacity:1"'

			this.strElemId := UINT_TO_STRING(i);

			hmi.in.cmd.draw.strStyle := 'id="3';

			styleStringGeneration;

			// DRAW SELECTED SHAPE WITH SPECIFIED PARAMETERS ON THE OVERLAY
			CASE hmi.in.cmd.draw.intShape OF
				0: // Rectangle
					brdkViGeom_drawSvgRectFromCP(this.tmp2D,hmi.in.cmd.draw.length,hmi.in.cmd.draw.width,hmi.in.cmd.draw.invRotation,ADR(hmi.out.svgOverlay),ADR(hmi.in.cmd.draw.strStyle));
				1: // Circle
					brdkViGeom_drawSvgCircle(this.tmp2D,hmi.in.cmd.draw.radius,ADR(hmi.out.svgOverlay),ADR(hmi.in.cmd.draw.strStyle));
				2: // Triangle
					brdkViGeom_drawSvgTriFromCP(this.tmp2D,hmi.in.cmd.draw.length,hmi.in.cmd.draw.width,hmi.in.cmd.draw.invRotation,ADR(hmi.out.svgOverlay),ADR(hmi.in.cmd.draw.strStyle));

			END_CASE;
		END_FOR;
	END_IF;

(*	//MEASUREMENT

	IF hwInstance[4].VF.measurement.in.common.numResults > 0 THEN

		hmi.out.svgOverlay := '';

		FOR i:= 1 TO hw.VF.measurement.in.common.numResults BY 1 DO
			this.tmp2D.x := DINT_TO_REAL(hw.VF.measurement.in.results[i-1].positionX) / 100.0;
			this.tmp2D.y := DINT_TO_REAL(hw.VF.measurement.in.results[i-1].positionY) / 100.0;

			// Style string generation
			// e.g.:'id="13" style="fill:blue;stroke:blue;stroke-width:5;fill-opacity:0.3;stroke-opacity:1"'

			this.strElemId := UINT_TO_STRING(i);

			hmi.in.cmd.draw.strStyle := 'id="4';

			styleStringGeneration;

			// DRAW SELECTED SHAPE WITH SPECIFIED PARAMETERS ON THE OVERLAY
			CASE hmi.in.cmd.draw.intShape OF
				0: // Rectangle
					brdkViGeom_drawSvgRectFromCP(this.tmp2D,hmi.in.cmd.draw.length,hmi.in.cmd.draw.width,hmi.in.cmd.draw.invRotation,ADR(hmi.out.svgOverlay),ADR(hmi.in.cmd.draw.strStyle));
				1: // Circle
					brdkViGeom_drawSvgCircle(this.tmp2D,hmi.in.cmd.draw.radius,ADR(hmi.out.svgOverlay),ADR(hmi.in.cmd.draw.strStyle));
				2: // Triangle
					brdkViGeom_drawSvgTriFromCP(this.tmp2D,hmi.in.cmd.draw.length,hmi.in.cmd.draw.width,hmi.in.cmd.draw.invRotation,ADR(hmi.out.svgOverlay),ADR(hmi.in.cmd.draw.strStyle));

			END_CASE;
		END_FOR;
	END_IF;
	*)

	//OCR

	IF hwInstance[5].VF.ocr.in.common.numResults > 0 THEN

		hmi.out.svgOverlay := '';

		FOR i:= 1 TO hw.VF.ocr.in.common.numResults BY 1 DO
			this.tmp2D.x := DINT_TO_REAL(hw.VF.ocr.in.results[i-1].positionX) / 100.0;
			this.tmp2D.y := DINT_TO_REAL(hw.VF.ocr.in.results[i-1].positionY) / 100.0;

			// Style string generation
			// e.g.:'id="13" style="fill:blue;stroke:blue;stroke-width:5;fill-opacity:0.3;stroke-opacity:1"'

			this.strElemId := UINT_TO_STRING(i);

			hmi.in.cmd.draw.strStyle := 'id="5';

			styleStringGeneration;

			hmi.in.cmd.draw.rotation:= hw.VF.ocr.in.results[i-1].orientation / 100.0;
			hmi.in.cmd.draw.invRotation:= -(hmi.in.cmd.draw.rotation);

			// DRAW SELECTED SHAPE WITH SPECIFIED PARAMETERS ON THE OVERLAY
			CASE hmi.in.cmd.draw.intShape OF
				0: // Rectangle
					brdkViGeom_drawSvgRectFromCP(this.tmp2D,hmi.in.cmd.draw.length,hmi.in.cmd.draw.width,hmi.in.cmd.draw.invRotation,ADR(hmi.out.svgOverlay),ADR(hmi.in.cmd.draw.strStyle));
				1: // Circle
					brdkViGeom_drawSvgCircle(this.tmp2D,hmi.in.cmd.draw.radius,ADR(hmi.out.svgOverlay),ADR(hmi.in.cmd.draw.strStyle));
				2: // Triangle
					brdkViGeom_drawSvgTriFromCP(this.tmp2D,hmi.in.cmd.draw.length,hmi.in.cmd.draw.width,hmi.in.cmd.draw.invRotation,ADR(hmi.out.svgOverlay),ADR(hmi.in.cmd.draw.strStyle));

			END_CASE;
		END_FOR;
	END_IF;

	//PIXEL COUNT

	IF hwInstance[6].VF.pixelCnt.in.common.numResults > 0 THEN

		hmi.out.svgOverlay := '';

		FOR i:= 1 TO hw.VF.pixelCnt.in.common.numResults BY 1 DO
			this.tmp2D.x := DINT_TO_REAL(hw.VF.pixelCnt.in.results[i-1].positionX) / 100.0;
			this.tmp2D.y := DINT_TO_REAL(hw.VF.pixelCnt.in.results[i-1].positionY) / 100.0;

			// Style string generation
			// e.g.:'id="13" style="fill:blue;stroke:blue;stroke-width:5;fill-opacity:0.3;stroke-opacity:1"'

			this.strElemId := UINT_TO_STRING(i);

			hmi.in.cmd.draw.strStyle := 'id="6';

			styleStringGeneration;

			// DRAW SELECTED SHAPE WITH SPECIFIED PARAMETERS ON THE OVERLAY
			CASE hmi.in.cmd.draw.intShape OF
				0: // Rectangle
					brdkViGeom_drawSvgRectFromCP(this.tmp2D,hmi.in.cmd.draw.length,hmi.in.cmd.draw.width,hmi.in.cmd.draw.invRotation,ADR(hmi.out.svgOverlay),ADR(hmi.in.cmd.draw.strStyle));
				1: // Circle
					brdkViGeom_drawSvgCircle(this.tmp2D,hmi.in.cmd.draw.radius,ADR(hmi.out.svgOverlay),ADR(hmi.in.cmd.draw.strStyle));
				2: // Triangle
					brdkViGeom_drawSvgTriFromCP(this.tmp2D,hmi.in.cmd.draw.length,hmi.in.cmd.draw.width,hmi.in.cmd.draw.invRotation,ADR(hmi.out.svgOverlay),ADR(hmi.in.cmd.draw.strStyle));

			END_CASE;
		END_FOR;
	END_IF;

END_ACTION
```

#### styleStringGeneration.st
```iecst
ACTION styleStringGeneration:

	brsstrcat(ADR(hmi.in.cmd.draw.strStyle),ADR(this.strElemId));					// string for element id attribute (value)
	brsstrcat(ADR(hmi.in.cmd.draw.strStyle),ADR('" style="'));						// string for beginning of the style paramateres (text)
	brsstrcat(ADR(hmi.in.cmd.draw.strStyle),ADR(hmi.in.cmd.draw.strFillColor));		// string for fill color attribute (text + value)

	IF i=hmi.in.cmd.intElemId THEN
	  	brsstrcat(ADR(hmi.in.cmd.draw.strStyle),ADR(';stroke:white'));
	ELSE
		brsstrcat(ADR(hmi.in.cmd.draw.strStyle),ADR(hmi.in.cmd.draw.strStrokeColor));	// string for stroke color attribute (text + value)
	END_IF;

	brsstrcat(ADR(hmi.in.cmd.draw.strStyle),ADR(';stroke-width:')); 				// string for stroke width attribute (text)
	brsstrcat(ADR(hmi.in.cmd.draw.strStyle),ADR(hmi.in.cmd.draw.strStrokeWidth));	// string for stroke width attribute (value)
	brsstrcat(ADR(hmi.in.cmd.draw.strStyle),ADR(';fill-opacity:')); 				// string for fill opacity attribute (text)
	brsstrcat(ADR(hmi.in.cmd.draw.strStyle),ADR(hmi.in.cmd.draw.strFillOpac)); 		// string for fill opacity attribute (value)
	brsstrcat(ADR(hmi.in.cmd.draw.strStyle),ADR(';stroke-opacity:')); 				// string for stroke opacity attribute (text)
	brsstrcat(ADR(hmi.in.cmd.draw.strStyle),ADR(hmi.in.cmd.draw.strStrokeOpac)); 	// string for stroke opacity attribute (value)

	brsstrcat(ADR(hmi.in.cmd.draw.strStyle),ADR('"'));

END_ACTION
```

#### tableResultsAction.st
```iecst
ACTION tableResultsAction:
	IF hw.VF.blob.in.common.numResults > 0 THEN
	  	FOR p:=0 TO hw.VF.ocr.in.common.numResults-1 DO
			hmi.out.VF.blob.ModelNumber[p+1] := hw.VF.blob.in.results[p].modelNumber;
			hmi.out.VF.blob.Clipped[p+1] := hw.VF.blob.in.results[p].clipped;
			hmi.out.VF.blob.Area[p+1] := hw.VF.blob.in.results[p].area;
			hmi.out.VF.blob.PositionX[p+1] := hw.VF.blob.in.results[p].positionX;
			hmi.out.VF.blob.PositionY[p+1] := hw.VF.blob.in.results[p].positionY;
			hmi.out.VF.blob.Orientation[p+1] := hw.VF.blob.in.results[p].orientation;
			hmi.out.VF.blob.MeanGrayValue[p+1] := hw.VF.blob.in.results[p].meanGreyValue;
			hmi.out.VF.blob.Length[p+1] := hw.VF.blob.in.results[p].length;
			hmi.out.VF.blob.Width[p+1] := hw.VF.blob.in.results[p].width;
		END_FOR;
	END_IF;

	IF hw.VF.codeReader.in.common.numResults > 0 THEN
		FOR p:=0 TO hw.VF.codeReader.in.common.numResults-1 DO
			hmi.out.VF.codeReader.CodeType[p+1] := hw.VF.codeReader.in.results[p].symbolType;
			hmi.out.VF.codeReader.Grading[p+1] := hw.VF.codeReader.in.results[p].gradingValue;
			hmi.out.VF.codeReader.PositionX[p+1] := hw.VF.codeReader.in.results[p].positionX;
			hmi.out.VF.codeReader.PositionY[p+1] := hw.VF.codeReader.in.results[p].positionY;
			hmi.out.VF.codeReader.Orientation[p+1] := hw.VF.codeReader.in.results[p].orientation;
		END_FOR;
	END_IF;

	IF hw.VF.matching.in.common.numResults > 0 THEN
		FOR p:=0 TO hw.VF.matching.in.common.numResults-1 DO
			hmi.out.VF.match.ModelNumber[p+1] := hw.VF.matching.in.results[p].modelNumber;
			hmi.out.VF.match.Score[p+1] := hw.VF.matching.in.results[p].score;
			hmi.out.VF.match.PositionX[p+1] := hw.VF.matching.in.results[p].positionX;
			hmi.out.VF.match.PositionY[p+1] := hw.VF.matching.in.results[p].positionY;
			hmi.out.VF.match.Orientation[p+1] := hw.VF.matching.in.results[p].orientation;
			hmi.out.VF.match.Scale[p+1] := hw.VF.matching.in.results[p].scale;
		END_FOR;
	END_IF;

	IF hw.VF.measurement.in.common.numResults > 0 THEN
		FOR p:=0 TO hw.VF.measurement.in.common.numResults-1 DO
			hmi.out.VF.measurement.Result[p+1] := hw.VF.measurement.in.results[p].result;
		END_FOR;
	END_IF;

	IF hw.VF.ocr.in.common.numResults > 0 THEN
		FOR p:=0 TO hw.VF.ocr.in.common.numResults-1 DO
			hmi.out.VF.ocr.Grading[p+1] := hw.VF.ocr.in.results[p].gradingValue;
			hmi.out.VF.ocr.PositionX[p+1] := hw.VF.ocr.in.results[p].positionX;
			hmi.out.VF.ocr.PositionY[p+1] := hw.VF.ocr.in.results[p].positionY;
			hmi.out.VF.ocr.Orientation[p+1] := hw.VF.ocr.in.results[p].orientation;
		END_FOR;
	END_IF;

	IF hw.VF.pixelCnt.in.common.numResults > 0 THEN
		FOR p:=0 TO hw.VF.pixelCnt.in.common.numResults-1 DO
			hmi.out.VF.pixelCnt.ModelNumber[p+1] := hw.VF.pixelCnt.in.results[p].modelNumber;
			hmi.out.VF.pixelCnt.ModelArea[p+1] := hw.VF.pixelCnt.in.results[p].modelArea;
			hmi.out.VF.pixelCnt.NumPixels[p+1] := hw.VF.pixelCnt.in.results[p].numPixels;
			hmi.out.VF.pixelCnt.MinGray[p+1] := hw.VF.pixelCnt.in.results[p].minGray;
			hmi.out.VF.pixelCnt.MaxGray[p+1] := hw.VF.pixelCnt.in.results[p].maxGray;
			hmi.out.VF.pixelCnt.DeviationGray[p+1] := hw.VF.pixelCnt.in.results[p].deviationGray;
			hmi.out.VF.pixelCnt.NumConnectedComponents[p+1] := hw.VF.pixelCnt.in.results[p].numConnectedComponents;
			hmi.out.VF.pixelCnt.PositionX[p+1] := hw.VF.pixelCnt.in.results[p].positionX;
			hmi.out.VF.pixelCnt.PositionY[p+1] := hw.VF.pixelCnt.in.results[p].positionY;
		END_FOR;
	END_IF;

END_ACTION
```

#### LocalFunctions.fun - not listed in the package file held
```iecst
FUNCTION_BLOCK VaGetList
	VAR_INPUT
		Enable : BOOL;
	END_VAR
	VAR_OUTPUT
		VaApplicationCnt : USINT;
		VaApplicationNames : ARRAY[0..MAX_IDX_VA_LIST] OF STRING[40];
		Status : UINT;
	END_VAR
	VAR
		State : USINT;
	END_VAR
	VAR CONSTANT
		STATE_WAIT : USINT := 0;
		STATE_NEXT_OBJ : USINT := 1;
		STATE_VA_NAME : USINT := 2;
	END_VAR
	VAR
		i : UINT;
		j : UINT;
		PrevIndex : UINT;
		ModuleList : MO_List_typ;
		ModuleStatus : UINT;
		zzEdge00000 : BOOL;
	END_VAR
END_FUNCTION_BLOCK

FUNCTION CrosshairDetailsText : BOOL
	VAR_INPUT
		strTarget : UDINT;
		strText : UDINT;
		fValue : REAL;
	END_VAR
	VAR
		tmpStr : STRING[50];
	END_VAR
END_FUNCTION

FUNCTION String2DataProvider : BOOL
	VAR_INPUT
		SourceString : UDINT;
		TargetString : UDINT;
	END_VAR
END_FUNCTION
```

#### Actions.st - not listed in the package file held
```iecst
ACTION ACTION_InitCodeTypes:
	CodeTypes[0]	:= 'Auto Identify (0)';;
	CodeTypes[1]	:= '2/5 Industrial (1)';
	CodeTypes[2]	:= '2/5 Interleaved (2)';
	CodeTypes[3]	:= 'Codebar (3)';
	CodeTypes[4]	:= 'Code 32 (4)';
	CodeTypes[5]	:= 'Code 39 (5)';
	CodeTypes[6]	:= 'Code 93 (6)';
	CodeTypes[7]	:= 'Code 128 (7)';
	CodeTypes[8]	:= 'MSI (8)';
	CodeTypes[9]	:= 'PharmaCode (9)';
	CodeTypes[10]	:= 'EAN-8 (10)';
	CodeTypes[11]	:= 'EAN-8 Add-On 2 (11)';
	CodeTypes[12]	:= 'EAN-8 Add-On 5 (12)';
	CodeTypes[13]	:= 'EAN-13 (13)';
	CodeTypes[14]	:= 'EAN-13 Add-On 2 (14)';
	CodeTypes[15]	:= 'EAN-13 Add-On 5 (15)';
	CodeTypes[20]	:= 'UPC-A (20)';
	CodeTypes[21]	:= 'UPC-A Add-On 2 (21)';
	CodeTypes[22]	:= 'UPC-A Add-On 5 (22)';
	CodeTypes[23]	:= 'UPC-E (23)';
	CodeTypes[24]	:= 'UPC-E Add-On 2 (24)';
	CodeTypes[25]	:= 'UPC-E Add-On 5 (25)';
	CodeTypes[30]	:= 'GS1-128 (30)';
	CodeTypes[31]	:= 'GS1 DataBar Omnidirectional (31)';
	CodeTypes[32]	:= 'GS1 DataBar Truncated (32)';
	CodeTypes[33]	:= 'GS1 DataBar Stacked (33)';
	CodeTypes[34]	:= 'GS1 DataBar Stacked Omnidirectional (34)';
	CodeTypes[35]	:= 'GS1 DataBar Limited (35)';
	CodeTypes[36]	:= 'GS1 DataBar Expanded (36)';
	CodeTypes[37]	:= 'GS1 DataBar ExpandedStacked (37)';
	CodeTypes[50]	:= 'Data Matrix ECC200 (50)';
	CodeTypes[51]	:= 'QR Code Model 1 (51)';
	CodeTypes[52]	:= 'QR Code Model 2 (52)';
	CodeTypes[53]	:= 'Micro QRCode (53)';
	CodeTypes[54]	:= 'PDF417 (54)';
	CodeTypes[55]	:= 'Aztec Code (55)';
	CodeTypes[60]	:= 'GS1 Data Matrix (60)';
	CodeTypes[61]	:= 'GS1 QR Code Model 1 (61)';
	CodeTypes[62]	:= 'GS1 QR Code Model 2 (62)';
	CodeTypes[63]	:= 'GS1 Aztec Code (63)';
	FOR i := 0 TO MAX_NUM_CODETYPES DO
		IF CodeTypes[i] <> '' THEN
			brsstrcat(ADR(visCodeTypePresentDropDownValues[i]), ADR('{"value":"'));
			brsitoa(i, ADR(tmpStr1));
			brsstrcat(ADR(visCodeTypePresentDropDownValues[i]), ADR(tmpStr1));
			brsstrcat(ADR(visCodeTypePresentDropDownValues[i]), ADR('","text":"'));
			brsstrcat(ADR(visCodeTypePresentDropDownValues[i]), ADR(CodeTypes[i]));
			brsstrcat(ADR(visCodeTypePresentDropDownValues[i]), ADR('"}'));
		END_IF
	END_FOR
END_ACTION
```

#### LocalFunctions.st - not listed in the package file held
```iecst
//******************************************************************************************************
// Create crosshair text
//******************************************************************************************************
FUNCTION CrosshairDetailsText
	tmpStr:= '<tspan class="text" x="10" dy="32">';
	brsstrcat(strTarget, ADR(tmpStr));
	brsstrcat(strTarget, strText);
	brsftoa(fValue, ADR(tmpStr));
	brsstrcat(strTarget, ADR(tmpStr));
	brsstrcat(strTarget, ADR('</tspan> '));

	CrosshairDetailsText := TRUE;
END_FUNCTION

//******************************************************************************************************
// Create mappView data provider string
//******************************************************************************************************
FUNCTION String2DataProvider
	brsstrcpy(TargetString, ADR('{"value":"'));
	brsstrcat(TargetString, SourceString);
	brsstrcat(TargetString, ADR('","text":"'));
	brsstrcat(TargetString, SourceString);
	brsstrcat(TargetString, ADR('"}'));
	String2DataProvider := TRUE;
END_FUNCTION

//******************************************************************************************************
// Create vision application list
//******************************************************************************************************
FUNCTION_BLOCK VaGetList
	IF (NOT Enable) THEN
		State := STATE_WAIT;
	END_IF

	CASE State OF
		// ----------------------------------------------------------------------------------------
		// Wait state
		STATE_WAIT:
			Status := ERR_FUB_ENABLE_FALSE;

			// Start new list
			IF EDGEPOS(Enable) THEN
				Status := ERR_FUB_BUSY;
				VaApplicationCnt := 0;
				PrevIndex := 16#FFFF;
				State := STATE_NEXT_OBJ;
				brsmemset(ADR(VaApplicationCnt),0, SIZEOF(VaApplicationCnt));
			END_IF
			// ----------------------------------------------------------------------------------------
		// Get next module
		STATE_NEXT_OBJ:
			// Get next module
			ModuleStatus := MO_list(PrevIndex,ADR(PrevIndex),ADR(ModuleList));

			// ----------------------------------------------------------------------------------------
			// OK
			IF ModuleStatus = ERR_OK AND ModuleList.type = 16#88 THEN
				State := STATE_VA_NAME;
			// ----------------------------------------------------------------------------------------
			// Last module reached
			ELSIF ModuleStatus = ERR_BUR_NOENTRY THEN
				Status := ERR_OK;
				State := STATE_WAIT;
			// ----------------------------------------------------------------------------------------
			// Error
			ELSIF ModuleStatus <> ERR_OK THEN
				Status := ModuleStatus;
				State := STATE_WAIT;
			END_IF
		// ----------------------------------------------------------------------------------------
		// Find vision application anme
		STATE_VA_NAME:
			FOR i:=0 TO 400 DO
				IF (brsmemcmp(ModuleList.adress+i, ADR('" Type="visionapplication"'), SIZEOF('" Type="visionapplication"')-1) = 0) THEN
					FOR j:=i-1 TO 1 BY -1 DO
						IF (brsmemcmp(ModuleList.adress+j, ADR('"'), SIZEOF('"')-1) = 0) THEN
							brsmemcpy(ADR(VaApplicationNames[VaApplicationCnt]), ModuleList.adress+j+1, i-j-1);
							VaApplicationCnt := VaApplicationCnt + 1;
							// Make sure we dont exceed array limit
							IF VaApplicationCnt > MAX_IDX_VA_LIST THEN
								Status := ERR_VA_LIST_NUM;
								State := STATE_WAIT;
								EXIT;
							END_IF
							EXIT;
						END_IF
					END_FOR
					EXIT;
				END_IF
			END_FOR
			State := STATE_NEXT_OBJ;
	END_CASE

END_FUNCTION_BLOCK
```

### Program Logical/Vision/Vi_visu (IEC)

#### Main.st - Init, cyclic, exit code
```iecst
// --------------------------------------------------------------------------------------------------------------------
// This is a support task for the mappView visualization. The following functions are implemneted
// - Disable mappView functions when camera is not ready, available
// - Transfer parameters after vision setup
// Version 2.x (Check revision history for details)
// --------------------------------------------------------------------------------------------------------------------
PROGRAM _INIT
	// -----------------------------------------------------------------------------------------------------------
	// Map global structure to local reference
	VisionSensor ACCESS ADR(gVisionSensor[gSelectedSensor]);
	Blob ACCESS ADR(tmpBlob);
	CodeReader ACCESS ADR(tmpCodeReader);
	Match ACCESS ADR(tmpMatch);
	MT ACCESS ADR(tmpMT);
	OCR ACCESS ADR(tmpOCR);
	Pixel ACCESS ADR(tmpPixel);

	// Map global structure to local reference
	VisionLight ACCESS ADR(gVisionLight[gSelectedLight]);

	// -----------------------------------------------------------------------------------------------------------
	// Preload code types
	FOR i := 0 TO MAX_NUM_CODETYPES DO
		IF CodeTypes[i] <> '' THEN
			brsstrcat(ADR(visCodeTypePresentDropDownValues[i]), ADR('{"value":"'));
			brsitoa(i, ADR(tmpStr1));
			brsstrcat(ADR(visCodeTypePresentDropDownValues[i]), ADR(tmpStr1));
			brsstrcat(ADR(visCodeTypePresentDropDownValues[i]), ADR('","text":"'));
			brsstrcat(ADR(visCodeTypePresentDropDownValues[i]), ADR(CodeTypes[i]));
			brsstrcat(ADR(visCodeTypePresentDropDownValues[i]), ADR('"}'));
		END_IF
	END_FOR

	// -----------------------------------------------------------------------------------------------------------
	visTableNo;
	InitialSearchSensor := TRUE;
	InitialSearchLight := TRUE;
END_PROGRAM

// -----------------------------------------------------------------------------------------------------------
// Cyclic part
// -----------------------------------------------------------------------------------------------------------
PROGRAM _CYCLIC
	// Select first available camera after reboot
	IF InitialSearchSensor THEN
		FOR i := 1 TO MAX_NUM_CAMS DO
			IF gVisionSensor[i].HW.Connected THEN
				gSelectedSensor := i;
				InitialSearchSensor := FALSE;
				EXIT;
			END_IF
		END_FOR
	END_IF

	// -----------------------------------------------------------------------------------------------------------
	// Map global structure to local reference for mappView
	// -----------------------------------------------------------------------------------------------------------
	// Make sure we dont exceed array limit
	IF(gSelectedSensor > MAX_NUM_CAMS) THEN
		gSelectedSensor := 1;
	END_IF
	IF(gSelectedSensor < 1) THEN
		gSelectedSensor := MAX_NUM_CAMS;
	END_IF

	// Assign pointers
	VisionSensor ACCESS ADR(gVisionSensor[gSelectedSensor]);
	IF(VisionSensor.CFG.DataStructure <> 0) THEN
		CASE VisionSensor.CFG.VisionFunction OF
			enumBlob:			Blob ACCESS VisionSensor.CFG.DataStructure;
			enumCoderReader:	CodeReader ACCESS VisionSensor.CFG.DataStructure;
			enumMatch:			Match ACCESS VisionSensor.CFG.DataStructure;
			enumMeasurement:	MT ACCESS VisionSensor.CFG.DataStructure;
			enumOCR:			OCR ACCESS VisionSensor.CFG.DataStructure;
			enumPixelCounter:	Pixel ACCESS VisionSensor.CFG.DataStructure;
		END_CASE
	ELSE
		RETURN;
	END_IF

	// Display camera status
	visCameraStatus := VisionSensor.DAT.StatusText;

	// -----------------------------------------------------------------------------------------------------------
	// Code Reader - selected/detected types
	// -----------------------------------------------------------------------------------------------------------
	IF VisionSensor.CFG.VisionFunction = enumCoderReader THEN
		IF visSelectedCodeType <> visSelectedCodeTypeOld THEN
			CodeReader.CodeType := UDINT_TO_USINT(brsatoi(ADR(visSelectedCodeType)));
		ELSE
			brsitoa(CodeReader.CodeType, ADR(visSelectedCodeType));
		END_IF
		visSelectedCodeTypeOld := visSelectedCodeType;
		IF visSelectedParameterMode <> visSelectedParameterModeOld THEN
			CodeReader.ParameterMode := UDINT_TO_USINT(brsatoi(ADR(visSelectedParameterMode)));
		ELSE
			brsitoa(CodeReader.ParameterMode, ADR(visSelectedParameterMode));
		END_IF
		visSelectedParameterModeOld := visSelectedParameterMode;
		FOR i := 1 TO MAX_NUM_RESULTS DO
			IF CodeReader.BarcodeType[i] <> 0 THEN
				brsstrcpy(ADR(visSelectedCodeTypeDetected[i]), ADR(CodeTypes[LIMIT(0, CodeReader.BarcodeType[i], MAX_NUM_CODETYPES)]));
			ELSE
				brsstrcpy(ADR(visSelectedCodeTypeDetected[i]), ADR(''));
			END_IF
		END_FOR
	END_IF

	// -----------------------------------------------------------------------------------------------------------
	// Translate flash color and segments from mappView to IO mapping
	// -----------------------------------------------------------------------------------------------------------
	IF visSensorFlashColor <> visSensorFlashColorOld THEN
		VisionSensor.DAT.FlashColor := UDINT_TO_USINT(brsatoi(ADR(visSensorFlashColor)));
	ELSE
		brsitoa(VisionSensor.DAT.FlashColor, ADR(visSensorFlashColor));
	END_IF
	visSensorFlashColorOld := visSensorFlashColor;
	IF brsmemcmp(ADR(visSelectedFlashSegment), ADR(visSelectedFlashSegmentOld), SIZEOF(visSelectedFlashSegment)) <> 0 THEN // The flash segments was changed in the mappView visualization
		VisionSensor.DAT.FlashSegment := SHL(visSelectedFlashSegment[0], 0) OR SHL(visSelectedFlashSegment[1], 1) OR SHL(visSelectedFlashSegment[2], 2) OR SHL(visSelectedFlashSegment[3], 3);
	ELSE
		visSelectedFlashSegment[0] := VisionSensor.DAT.FlashSegment.0;
		visSelectedFlashSegment[1] := VisionSensor.DAT.FlashSegment.1;
		visSelectedFlashSegment[2] := VisionSensor.DAT.FlashSegment.2;
		visSelectedFlashSegment[3] := VisionSensor.DAT.FlashSegment.3;
	END_IF
	visSelectedFlashSegmentOld := visSelectedFlashSegment;

	// -----------------------------------------------------------------------------------------------------------
	// Disable command buttons when camera is disconnected, not ready, processing an image or vision cockpit is open
	// -----------------------------------------------------------------------------------------------------------
	IF(NOT VisionSensor.HW.Connected OR NOT VisionSensor.HW.Ready OR VisionSensor.DAT.ImageProcessingActive OR VisionSensor.DAT.CockpitIsActive) THEN
		visSensorEnableCommand := FALSE;
	ELSE
		visSensorEnableCommand := TRUE;
	END_IF

	// -----------------------------------------------------------------------------------------------------------
	// Disable setup buttons when camera is disconnected, processing an image or not ready
	// -----------------------------------------------------------------------------------------------------------
	IF(NOT VisionSensor.HW.Connected OR NOT (VisionSensor.HW.Ready OR AutoSetupRunning[gSelectedSensor]) OR VisionSensor.DAT.ImageProcessingActive) THEN
		visEnableSetup := FALSE;
	ELSE
		visEnableSetup := TRUE;
	END_IF

	// -----------------------------------------------------------------------------------------------------------
	// Fire trigger for camera image
	// -----------------------------------------------------------------------------------------------------------
	IF((visImageTrigger OR EDGEPOS(VisionSensor.DAT.Enable)) AND VisionSensor.HW.Ready AND NOT VisionSensor.DAT.ImageProcessingActive) THEN
		// Add default delay and fire trigger
		IF NETTIME_ENABLE THEN
			VisionSensor.DAT.NettimeDelay := NettimeCurrent_us + NETTIME_DEFAULT_DELAY;
		END_IF
		// Hide previous results
		FOR i := 1 TO MAX_NUM_RESULTS DO
			visCrossHair.SvgVisible[i] := FALSE;
		END_FOR;
		VisionSensor.CMD.ImageTrigger	:= TRUE;
		visImageTrigger					:= FALSE;
		VisionSensor.DAT.Active			:= TRUE;
	END_IF

	// -----------------------------------------------------------------------------------------------------------
	// Get image from camera
	// -----------------------------------------------------------------------------------------------------------
	IF EDGENEG(VisionSensor.CMD.ImageTrigger) THEN
		gVisionImage.CFG.ComponentLink := gVisionSensor[gSelectedSensor].CFG.ComponentLink;
		gVisionImage.CMD.GetImage := TRUE;
	END_IF

	// -----------------------------------------------------------------------------------------------------------
	// Repetitive mode
	// -----------------------------------------------------------------------------------------------------------
	visEnableRepetitive := visSensorEnableCommand OR visRepetitiveMode;
	IF visRepetitiveMode THEN
		RepetitiveModeTimer.IN := TRUE;
		IF RepetitiveModeTimer.Q THEN
			IF VisionSensor.HW.Ready AND NOT VisionSensor.DAT.ImageProcessingActive THEN
				IF NETTIME_ENABLE THEN
					VisionSensor.DAT.NettimeDelay := NettimeCurrent_us + NETTIME_DEFAULT_DELAY;
				END_IF
				RepetitiveModeTimer.IN := FALSE;
				VisionSensor.CMD.ImageTrigger := TRUE;
			END_IF
		END_IF
		VisionSensor.DAT.Enable := FALSE;
	ELSE
		RepetitiveModeTimer.IN := TRUE;
	END_IF
	RepetitiveModeTimer(PT := T#3000ms);

	// -----------------------------------------------------------------------------------------------------------
	// Select first available light after reboot
	// -----------------------------------------------------------------------------------------------------------
	IF InitialSearchLight THEN
		FOR i := 1 TO MAX_NUM_LIGHTS DO
			IF gVisionLight[i].HW.Connected THEN
				gSelectedLight := i;
				InitialSearchLight := FALSE;
				EXIT;
			END_IF
		END_FOR
	END_IF

	// -----------------------------------------------------------------------------------------------------------
	// Map global structure to local reference
	// -----------------------------------------------------------------------------------------------------------
	// Make sure we dont exceed array limit
	IF(gSelectedLight > MAX_NUM_LIGHTS) THEN
		gSelectedLight := 1;
	END_IF
	IF(gSelectedLight < 1) THEN
		gSelectedLight := MAX_NUM_LIGHTS;
	END_IF
	VisionLight ACCESS ADR(gVisionLight[gSelectedLight]);

	// -----------------------------------------------------------------------------------------------------------
	// Translate flash color from mappView to IO mapping
	// -----------------------------------------------------------------------------------------------------------
	// Hint: Normally copy from recipe (VisionLight) to visu. Only in case of a change in the visu copy to recipe
	IF visLightsFlashColor <> visLightsFlashColorOld THEN // The flash color was changed in the mappView visualization
		VisionLight.DAT.FlashColor := UDINT_TO_USINT(brsatoi(ADR(visLightsFlashColor)));
	ELSE
		brsitoa(VisionLight.DAT.FlashColor, ADR(visLightsFlashColor));
	END_IF
	visLightsFlashColorOld := visLightsFlashColor;

	// -----------------------------------------------------------------------------------------------------------
	// Reset Light trigger manually
	// -----------------------------------------------------------------------------------------------------------
	IF (visLightsReset) THEN
		VisionLight.CMD.FlashTrigger := FALSE;
		visLightsReset := FALSE;
	END_IF

	// -----------------------------------------------------------------------------------------------------------
	// Fire trigger for lights
	// -----------------------------------------------------------------------------------------------------------
	IF(visLightsTrigger AND VisionLight.HW.Ready) THEN
		// Add default delay and fire trigger
		IF NETTIME_ENABLE THEN
			VisionLight.DAT.NettimeDelay := NettimeCurrent_us + NETTIME_DEFAULT_DELAY;
		END_IF
		VisionLight.CMD.FlashTrigger := TRUE;
		visLightsTrigger := FALSE;
	END_IF

	// -----------------------------------------------------------------------------------------------------------
	// Disable command button when light is disconnected or not ready
	// -----------------------------------------------------------------------------------------------------------
	IF(NOT VisionLight.HW.Connected OR NOT VisionLight.HW.Ready) THEN
		visLightsEnableCommand := FALSE;
	ELSE
		visLightsEnableCommand := TRUE;
	END_IF

	// -----------------------------------------------------------------------------------------------------------
	// Enable fields for different light types
	// -----------------------------------------------------------------------------------------------------------
	visEnableLightBarValues := VisionLight.CFG.LightType = enumLightbar;

	// -----------------------------------------------------------------------------------------------------------
	// Draw cross hairs on main page
	// -----------------------------------------------------------------------------------------------------------
	IF (EDGENEG(gVisionImage.CMD.GetImage) AND visCrossHair.ShowCrosshair) OR EDGEPOS(visCrossHair.ShowCrosshair) OR (visCrossHair.DetailsNo <> DetailsNoOld) THEN
		// -----------------------------------------------------------------------------------------------------------
		// Handle details no
		IF(visCrossHair.DetailsNo < 1) THEN
			visCrossHair.DetailsNo := VisionSensor.DAT.ResultCnt;
		END_IF
		IF(visCrossHair.DetailsNo > VisionSensor.DAT.ResultCnt) THEN
			visCrossHair.DetailsNo := 1;
		END_IF
		IF visCrossHair.PixelRatio = 0 THEN
			RETURN;
		END_IF
		DetailsNoOld := visCrossHair.DetailsNo;
		brsmemset(ADR(gVisionImage.DAT.Crosshair), 0, SIZEOF(gVisionImage.DAT.Crosshair));

		// -----------------------------------------------------------------------------------------------------------
		// Create cross hairs and data for all results
		FOR i := 1 TO MAX_NUM_RESULTS DO
			visCrossHair.SvgTransformation[i] := '';
			visCrossHair.SvgVisible[i] := FALSE;
			CrosshairPositionX := 0;
			CrosshairPositionY := 0;
			gVisionImage.DAT.Crosshair[i].CrosshairX		:= 0;
			gVisionImage.DAT.Crosshair[i].CrosshairY		:= 0;
			gVisionImage.DAT.Crosshair[i].CrosshairRotate	:= 0;
			brsmemset(ADR(gVisionImage.DAT.Crosshair[i].Text), 0, SIZEOF(gVisionImage.DAT.Crosshair[i].Text));

			// -----------------------------------------------------------------------------------------------------------
			// Make sure we have data to display
			IF(VisionSensor.DAT.ResultCnt <> 0 AND i <= VisionSensor.DAT.ResultCnt) THEN
				// Select data source from vision function
				CASE VisionSensor.CFG.VisionFunction OF
					enumBlob:
						CrosshairModelNumber := gBlob.ModelNumber[i];
						CrosshairPositionX := UDINT_TO_REAL(gBlob.PositionX[i]);
						CrosshairPositionY := UDINT_TO_REAL(gBlob.PositionY[i]);
						CrosshairOrientation := gBlob.Orientation[i];
					enumMatch:
						CrosshairModelNumber := gMatch.ModelNumber[i];
						CrosshairPositionX := UDINT_TO_REAL(gMatch.PositionX[i]);
						CrosshairPositionY := UDINT_TO_REAL(gMatch.PositionY[i]);
						CrosshairOrientation := gMatch.Orientation[i];
					enumCoderReader:
						CrosshairPositionX := UDINT_TO_REAL(gCodeReader.PositionX[i]);
						CrosshairPositionY := UDINT_TO_REAL(gCodeReader.PositionY[i]);
						CrosshairOrientation := gCodeReader.Orientation[i];
					enumOCR:
						CrosshairPositionX := UDINT_TO_REAL(gOCR.PositionX[i]);
						CrosshairPositionY := UDINT_TO_REAL(gOCR.PositionY[i]);
						CrosshairOrientation := gOCR.Orientation[i];
					enumMeasurement:
						IF(gMT.UseResultAsXY = TRUE) THEN
							CrosshairPositionX := UDINT_TO_REAL(gMT.Result[i])/10;
							CrosshairPositionY := UDINT_TO_REAL(gMT.Result[i+1])/10;
							i := i + 1;
						END_IF
				END_CASE

				// -----------------------------------------------------------------------------------------------------------
				// Show crosshair except for measurement function
				IF (VisionSensor.CFG.VisionFunction <> enumMeasurement OR gMT.UseResultAsXY = TRUE) THEN
					// -----------------------------------------------------------------------------------------------------------
					// Set start values
					IF(CrosshairPositionX <> 0 AND CrosshairPositionY <> 0) THEN
						visCrossHair.SvgVisible[i] := TRUE;

						// Highlight selected crosshair and show detailed information
						IF(visCrossHair.DetailsNo = i) THEN
							tmpStr1 := '[{"select":"#CrosshairBlue","display":false}, {"select":"#CrosshairRed","display":true, "translate":[';
						ELSE
							tmpStr1 := '[{"select":"#CrosshairRed","display":false}, { "select":"#CrosshairBlue","display":true, "translate":[';
						END_IF

						// Calculate cross hair X offset
						tmpXI := CrosshairPositionX / visCrossHair.PixelRatio;
						tmpC := USINT_TO_REAL(visCrossHair.Size) * visCrossHair.Scale / 2.0;
						brsitoa(REAL_TO_INT(tmpXI - tmpC), ADR(tmpStr2));
						brsstrcat(ADR(tmpStr1), ADR(tmpStr2));
						brsstrcat(ADR(tmpStr1), ADR(','));
						gVisionImage.DAT.Crosshair[i].CrosshairX := tmpXI - tmpC;

						// Calculate cross hair Y offset
						tmpYI := CrosshairPositionY / visCrossHair.PixelRatio;
						brsitoa(REAL_TO_INT(tmpYI - tmpC), ADR(tmpStr2));
						brsstrcat(ADR(tmpStr1), ADR(tmpStr2));
						gVisionImage.DAT.Crosshair[i].CrosshairY := tmpYI - tmpC;

						// Add cross hair scaling
						brsstrcat(ADR(tmpStr1), ADR('],"scale":['));
						brsftoa(visCrossHair.Scale, ADR(tmpStr2));
						brsstrcat(ADR(tmpStr1), ADR(tmpStr2));
						brsstrcat(ADR(tmpStr1), ADR(','));
						brsftoa(visCrossHair.Scale, ADR(tmpStr2));
						brsstrcat(ADR(tmpStr1), ADR(tmpStr2));

						// Add cross hair rotation
						brsstrcat(ADR(tmpStr1), ADR('],"spin":['));
						brsftoa(CrosshairOrientation/-100, ADR(tmpStr2));
						brsstrcat(ADR(tmpStr1), ADR(tmpStr2));
						brsstrcat(ADR(tmpStr1), ADR(','));
						brsitoa(visCrossHair.Size/2, ADR(tmpStr2));
						brsstrcat(ADR(tmpStr1), ADR(tmpStr2));
						brsstrcat(ADR(tmpStr1), ADR(','));
						brsstrcat(ADR(tmpStr1), ADR(tmpStr2));
						brsstrcat(ADR(tmpStr1), ADR(']}]'));
						visCrossHair.SvgTransformation[i] := tmpStr1;
						gVisionImage.DAT.Crosshair[i].CrosshairRotate := CrosshairOrientation/-100;

						// -----------------------------------------------------------------------------------------------------------
						// Add text data to selected cross hair
						IF(visCrossHair.DetailsNo = i) THEN
							tmpStr1 := '<text class="cText" fill="red" font-size="22" font-family="Helvetica, Arial, sans-serif" x="';
						ELSE
							tmpStr1 := '<text class="cText" fill="blue" font-size="22" font-family="Helvetica, Arial, sans-serif" x="';
						END_IF
						brsitoa(REAL_TO_INT(tmpXI - tmpC + visCrossHair.Size), ADR(tmpStr2));
						brsstrcat(ADR(tmpStr1), ADR(tmpStr2));
						brsstrcat(ADR(tmpStr1), ADR('" y="'));
						brsitoa(REAL_TO_INT(tmpYI - tmpC + visCrossHair.Size/2), ADR(tmpStr2));
						brsstrcat(ADR(tmpStr1), ADR(tmpStr2));
						brsstrcat(ADR(tmpStr1), ADR('"> '));

						// Create prototype for new entry
						tmpStr3:= '<tspan class="text" x="';
						brsitoa(REAL_TO_INT(tmpXI + tmpC), ADR(tmpStr2));
						brsstrcat(ADR(tmpStr3), ADR(tmpStr2));
						brsstrcat(ADR(tmpStr3), ADR('" dy="-5" >'));

						// Add result no information
						brsstrcat(ADR(tmpStr1), ADR(tmpStr3));
						brsitoa(i, ADR(tmpStr2));
						brsstrcat(ADR(tmpStr1), ADR(tmpStr2));
						brsstrcat(ADR(tmpStr1), ADR('</tspan></text>'));

						IF(visCrossHair.DetailsNo = i) THEN
							// -----------------------------------------------------------------------------------------------------------
							// Add text data from selected cross hair
							brsstrcat(ADR(tmpStr1), ADR('<text class="cText" fill="red" font-size="35" font-family="Helvetica, Arial, sans-serif" x="10" y="10"> '));

							// Add modell ID information for blob and match
							IF(VisionSensor.CFG.VisionFunction = enumBlob OR VisionSensor.CFG.VisionFunction = enumMatch) THEN
								CrosshairDetailsText(ADR(tmpStr1),  ADR('ID: '), CrosshairModelNumber);
							END_IF
							// Add X and Y position information
							IF(CrosshairPositionX <> 0) THEN
								CrosshairDetailsText(ADR(tmpStr1),  ADR('Pos X: '), CrosshairPositionX/visCrossHair.PixelRatio);
							END_IF
							IF(CrosshairPositionY <> 0) THEN
								CrosshairDetailsText(ADR(tmpStr1),  ADR('Pos Y: '), CrosshairPositionY/visCrossHair.PixelRatio);
							END_IF
							// Add orientation information
							IF(VisionSensor.CFG.VisionFunction <> enumMeasurement) THEN
								CrosshairDetailsText(ADR(tmpStr1),  ADR('Orientation: '), CrosshairOrientation/visCrossHair.PixelRatio);
							END_IF
							// Add detail information for blob
							IF(VisionSensor.CFG.VisionFunction = enumBlob AND gBlob.EnhancedBlobInformation = 1) THEN
								CrosshairDetailsText(ADR(tmpStr1),  ADR('Clipped: '), gBlob.Clipped[i]);
								CrosshairDetailsText(ADR(tmpStr1),  ADR('Gray: '), gBlob.MeanGrayValue[i]);
								CrosshairDetailsText(ADR(tmpStr1),  ADR('Length: '), UDINT_TO_REAL(gBlob.Length[i])/visCrossHair.PixelRatio);
								CrosshairDetailsText(ADR(tmpStr1),  ADR('Width: '), UDINT_TO_REAL(gBlob.Width[i])/visCrossHair.PixelRatio);
								CrosshairDetailsText(ADR(tmpStr1),  ADR('Area: '), UDINT_TO_REAL(gBlob.Area[i])/visCrossHair.PixelRatio);
							END_IF
							// Add detail information for match
							IF(VisionSensor.CFG.VisionFunction = enumMatch) THEN
								CrosshairDetailsText(ADR(tmpStr1),  ADR('Score: '), gMatch.Score[i]);
								CrosshairDetailsText(ADR(tmpStr1),  ADR('Scale: '), gMatch.Scale[i]);
							END_IF
							// Add detail information for code reader
							IF(VisionSensor.CFG.VisionFunction = enumCoderReader) THEN
								//CrosshairDetailsText(ADR(tmpStr1),  ADR('Code:'), UDINT_TO_REAL(CodeReader.BarcodeType[i]));
								tmpStr2:= '<tspan class="text" x="10" dy="32">';
								brsstrcat(ADR(tmpStr1), ADR(tmpStr2));
								brsstrcat(ADR(tmpStr1), ADR('Code: '));
								brsstrcat(ADR(tmpStr1), ADR(CodeTypes[LIMIT(0, gCodeReader.BarcodeType[i], MAX_NUM_CODETYPES)]));
								brsstrcat(ADR(tmpStr1), ADR('</tspan> '));
							END_IF
							brsstrcat(ADR(tmpStr1), ADR('</text>'));
						END_IF
					END_IF
					// -----------------------------------------------------------------------------------------------------------
					// Add result information measurement
				ELSE
					visCrossHair.SvgTransformation[i] := '[{"select":"#CrosshairRed","display":false}, {"select":"#CrosshairBlue","display":false}]';
					visCrossHair.SvgVisible[i] := TRUE;
					brsstrcpy(ADR(tmpStr1), ADR('<text class="cText" fill="red" font-size="35" font-family="Helvetica, Arial, sans-serif" x="10" y="'));
					brsitoa(i*40, ADR(tmpStr2));
					brsstrcat(ADR(tmpStr1), ADR(tmpStr2));
					brsstrcat(ADR(tmpStr1), ADR('"> '));
					CrosshairDetailsText(ADR(tmpStr1),  ADR('Result:'), UDINT_TO_REAL(gMT.Result[i])/1000);
					brsstrcat(ADR(tmpStr1), ADR('</text>'));
				END_IF
				visCrossHair.SvgContent[i] := tmpStr1;
				// for saving svg file
				brsstrcpy(ADR(gVisionImage.DAT.Crosshair[i].Text), ADR(tmpStr1));
			END_IF
		END_FOR
	END_IF
END_PROGRAM
```

#### Types.typ - Local data types
```iecst
TYPE
	typCrossHair : 	STRUCT  (*Cross hair data structure*)
		SvgTransformation : ARRAY[1..MAX_NUM_RESULTS]OF STRING[200] := [10('')]; (*Transformation string for paper widget*)
		SvgContent : ARRAY[1..MAX_NUM_RESULTS]OF STRING[1000]; (*Transformation string for paper widget*)
		SvgVisible : ARRAY[1..MAX_NUM_RESULTS]OF BOOL := [10(FALSE)];
		Scale : REAL := 1; (*Scale size of the cross hair*)
		PixelRatio : REAL := 100; (*Position value for one pixel*)
		Size : USINT := 80; (*Size of the cross hair in pixel*)
		Font : USINT := 35;
		DetailsNo : USINT := 1;
		ShowCrosshair : BOOL := TRUE; (*Enable/Disable cross hairs*)
	END_STRUCT;
END_TYPE
```

#### Variables.var - Local variables
```iecst
(*-----------------------------------------------------------------------------------------------------------------------------------------*)
(*Main vision and data structures*)
VAR
	VisionSensor : REFERENCE TO typVisionMain; (*General vision functions that are independent from the inspection function*)
	VisionLight : REFERENCE TO typLightMain; (*General vision functions that are independent from the inspection function*)
	Match : REFERENCE TO typMatchMain; (*Data that is specific for the match function*)
	CodeReader : REFERENCE TO typCodeReaderMain; (*Data that is specific for the code reader*)
	MT : REFERENCE TO typMTMain; (*Data that is specific for the MT function*)
	OCR : REFERENCE TO typOCRMain; (*Data that is specific for the OCR function*)
	Blob : REFERENCE TO typBlobMain; (*Data that is specific for the blob function*)
	Pixel : REFERENCE TO typPixelMain; (*Data that is specific for the blob function*)
	tmpMatch : {REDUND_UNREPLICABLE} typMatchMain; (*Data that is specific for the match function*)
	tmpCodeReader : {REDUND_UNREPLICABLE} typCodeReaderMain; (*Data that is specific for the code reader*)
	tmpMT : {REDUND_UNREPLICABLE} typMTMain; (*Data that is specific for the OCR function*)
	tmpOCR : {REDUND_UNREPLICABLE} typOCRMain; (*Data that is specific for the OCR function*)
	tmpBlob : {REDUND_UNREPLICABLE} typBlobMain; (*Data that is specific for the blob function*)
	tmpPixel : {REDUND_UNREPLICABLE} typPixelMain; (*Data that is specific for the blob function*)
END_VAR
(*-----------------------------------------------------------------------------------------------------------------------------------------*)
(*Sensor variables*)
VAR
	visSensorEnableCommand : BOOL; (*Enable/Disable vision trigger and enable when camera is not ready*)
	visEnableSetup : BOOL; (*Enable/Disable vision setup when camera is not ready*)
	visEnableRepetitive : BOOL; (*Enable/Disable repetitive mode*)
	visImageTrigger : BOOL; (*Trigger new image*)
	visSensorFlashColor : STRING[10]; (*Flash color string*)
	visSensorFlashColorOld : STRING[10]; (*Flash color string*)
	visSelectedFlashSegment : ARRAY[0..3] OF USINT := [4(1)]; (*Selected flash segments*)
	visSelectedFlashSegmentOld : ARRAY[0..3] OF USINT := [4(1)]; (*Selected flash segments*)
	visRepetitiveMode : BOOL; (*Enable/Disable repetitive mode*)
	RepetitiveModeTimer : TON; (*Timer for repetitive mode*)
	InitialSearchSensor : BOOL; (*Flag for first boot*)
	AutoSetupRunning : ARRAY[1..MAX_NUM_CAMS] OF BOOL; (*Flag for auto setup running*)
END_VAR
(*-----------------------------------------------------------------------------------------------------------------------------------------*)
(*Lights variables*)
VAR
	InitialSearchLight : BOOL;
	visLightsTrigger : BOOL;
	visLightsReset : BOOL;
	visLightsEnableCommand : BOOL;
	visLightsFlashColor : STRING[10]; (*Flash color string*)
	visLightsFlashColorOld : STRING[10];
	visEnableLightBarValues : BOOL;
END_VAR
(*-----------------------------------------------------------------------------------------------------------------------------------------*)
(*Code Reader*)
VAR
	visSelectedCodeTypeDetected : ARRAY[1..MAX_NUM_RESULTS] OF STRING[80]; (*HMI helper string*)
	visSelectedCodeType : STRING[80]; (*HMI helper string*)
	visSelectedCodeTypeOld : STRING[80]; (*HMI helper string*)
	visSelectedParameterMode : STRING[80]; (*HMI helper string*)
	visSelectedParameterModeOld : STRING[80]; (*HMI helper string*)
	visCodeTypePresentDropDownValues : ARRAY[0..MAX_NUM_CODETYPES] OF STRING[80];
END_VAR
(*-----------------------------------------------------------------------------------------------------------------------------------------*)
(*Image, crosshair data and constants*)
VAR
	visCrossHair : typCrossHair; (*Data structure to draw the crosshairs on the main page*)
	CrosshairModelNumber : USINT;
	CrosshairPositionX : REAL;
	CrosshairPositionY : REAL;
	CrosshairOrientation : INT;
	tmpStr1 : STRING[1000];
	tmpStr2 : STRING[100];
	tmpStr3 : STRING[100];
	tmpC : REAL;
	tmpYI : REAL;
	tmpXI : REAL;
	DetailsNoOld : USINT;
	visTableNo : ARRAY[1..MAX_NUM_RESULTS] OF USINT := [1,2,3,4,5,6,7,8,9,10];
	i : UINT;
	visCameraStatus : STRING[30];
END_VAR
```

#### LocalFunctions.fun - Local function definition
```iecst
FUNCTION CrosshairDetailsText : BOOL
	VAR_INPUT
		strTarget : UDINT;
		strText : UDINT;
		fValue : REAL;
	END_VAR
	VAR
		tmpStr : STRING[50];
	END_VAR
END_FUNCTION

FUNCTION String2DataProvider : BOOL
	VAR_INPUT
		SourceString : UDINT;
		TargetString : UDINT;
	END_VAR
END_FUNCTION
```

#### LocalFunctions.st - Local function code
```iecst
//******************************************************************************************************
// Create crosshair text
//******************************************************************************************************
FUNCTION CrosshairDetailsText
	tmpStr:= '<tspan class="text" x="10" dy="32">';
	brsstrcat(strTarget, ADR(tmpStr));
	brsstrcat(strTarget, strText);
	brsftoa(fValue, ADR(tmpStr));
	brsstrcat(strTarget, ADR(tmpStr));
	brsstrcat(strTarget, ADR('</tspan> '));

	CrosshairDetailsText := TRUE;
END_FUNCTION

//******************************************************************************************************
// Create mappView data provider string
//******************************************************************************************************
FUNCTION String2DataProvider
	brsstrcpy(TargetString, ADR('{"value":"'));
	brsstrcat(TargetString, SourceString);
	brsstrcat(TargetString, ADR('","text":"'));
	brsstrcat(TargetString, SourceString);
	brsstrcat(TargetString, ADR('"}'));
	String2DataProvider := TRUE;
END_FUNCTION
```

### Program Logical/Vision/Vi_image (IEC)
